KUKA KRL program: MyProgram_195().src

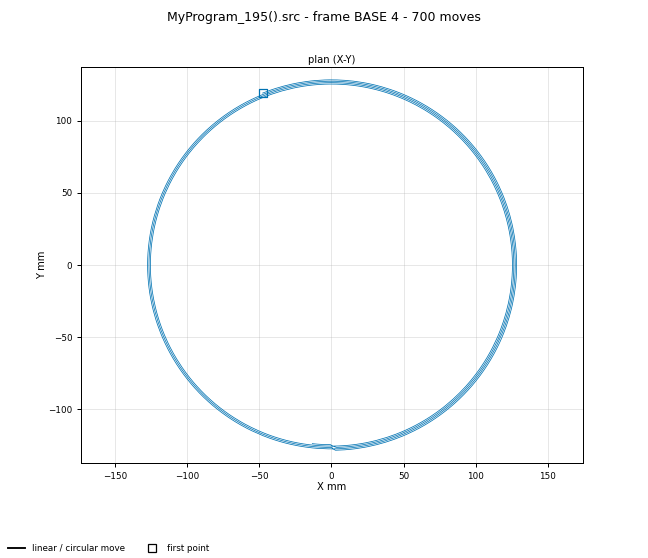
[picture p0: tool path of MyProgram_195().src in frame BASE 4, 700 of 700 moves have a stored position in this frame; points joined in program order, loops and branches not executed]
&ACCESS RVP
&REL 1
&PARAM TEMPLATE = C:\KRC\Roboter\Template\vorgabe
&PARAM EDITMASK = *
DEF MyProgram_195()
; ---- Setting reference (Base) ----
$BASE = BASE_DATA[4]

; --------------------------
; ---- Setting tool (TCP) ----
$TOOL = TOOL_DATA[3]
; --------------------------

$VEL.CP = VEL_APROX_PRINT
Startdeposition()
$VEL.CP = VEL_PRINT
LIN {X -47.6589,Y 119.2143,Z 141,A 107.4986,B 24.9483,C -1.6626,E1 24.9417,E2 698.8654} C_DIS
LIN {X -44.8255,Y 120.308,Z 141,A 106.1446,B 24.9481,C -1.6645,E1 24.9452,E2 700.2177} C_DIS
LIN {X -41.9136,Y 121.3531,Z 141,A 104.7349,B 24.9481,C -1.6649,E1 24.9489,E2 701.6293} C_DIS
LIN {X -38.7242,Y 122.4086,Z 141,A 103.221,B 24.948,C -1.666,E1 24.953,E2 703.1433} C_DIS
LIN {X -35.7429,Y 123.3121,Z 141,A 101.8617,B 24.9478,C -1.669,E1 24.9566,E2 704.4977} C_DIS
LIN {X -32.8744,Y 124.1073,Z 141,A 100.5283,B 24.9478,C -1.6702,E1 24.9602,E2 705.8304} C_DIS
LIN {X -29.3377,Y 124.9928,Z 141,A 98.9078,B 24.9476,C -1.672,E1 24.9646,E2 707.4487} C_DIS
LIN {X -26.9746,Y 125.5218,Z 141,A 97.7935,B 24.9476,C -1.6714,E1 24.9676,E2 708.5658} C_DIS
LIN {X -23.7646,Y 126.1693,Z 141,A 96.3869,B 24.9474,C -1.6752,E1 24.9714,E2 709.965} C_DIS
LIN {X -20.4905,Y 126.7435,Z 141,A 94.8925,B 24.9474,C -1.6758,E1 24.9756,E2 711.4594} C_DIS
LIN {X -17.7576,Y 127.1542,Z 141,A 93.4973,B 24.9478,C -1.6688,E1 24.9795,E2 712.8724} C_DIS
LIN {X -13.7906,Y 127.6448,Z 141,A 91.8165,B 24.9474,C -1.6748,E1 24.9841,E2 714.54} C_DIS
LIN {X -10.7812,Y 127.9341,Z 141,A 90.5046,B 24.9473,C -1.6773,E1 24.9877,E2 715.8467} C_DIS
LIN {X -7.5605,Y 128.1653,Z 141,A 89.0931,B 24.9472,C -1.6793,E1 24.9916,E2 717.254} C_DIS
LIN {X -4.6723,Y 128.3031,Z 141,A 87.7567,B 24.9472,C -1.6775,E1 24.9954,E2 718.5949} C_DIS
LIN {X -1.4217,Y 128.3818,Z 141,A 86.3404,B 24.9472,C -1.6795,E1 24.9993,E2 720.0065} C_DIS
LIN {X 3.8968,Y 128.329,Z 141,A 83.9462,B 24.9472,C -1.6789,E1 25.006,E2 722.4018} C_DIS
LIN {X 6.622,Y 128.2169,Z 141,A 82.776,B 24.947,C -1.6813,E1 25.0093,E2 723.5661} C_DIS
LIN {X 9.4027,Y 128.0429,Z 141,A 81.4527,B 24.9473,C -1.6773,E1 25.013,E2 724.8981} C_DIS
LIN {X 12.4041,Y 127.787,Z 141,A 80.1206,B 24.9473,C -1.6778,E1 25.0167,E2 726.2284} C_DIS
LIN {X 15.3395,Y 127.468,Z 141,A 78.7687,B 24.9473,C -1.6759,E1 25.0204,E2 727.5839} C_DIS
LIN {X 18.503,Y 127.0477,Z 141,A 77.424,B 24.9471,C -1.6794,E1 25.0241,E2 728.919} C_DIS
LIN {X 21.4719,Y 126.5797,Z 141,A 76.0524,B 24.9473,C -1.6774,E1 25.0279,E2 730.2939} C_DIS
LIN {X 25.2565,Y 125.8792,Z 141,A 74.2851,B 24.9475,C -1.6743,E1 25.0328,E2 732.0666} C_DIS
LIN {X 28.5721,Y 125.1677,Z 141,A 72.8026,B 24.9475,C -1.675,E1 25.0368,E2 733.5454} C_DIS
LIN {X 31.6188,Y 124.433,Z 141,A 71.4069,B 24.9475,C -1.6743,E1 25.0406,E2 734.9406} C_DIS
LIN {X 34.9234,Y 123.5467,Z 141,A 69.8932,B 24.9475,C -1.6739,E1 25.0447,E2 736.4528} C_DIS
LIN {X 37.9171,Y 122.661,Z 141,A 68.4959,B 24.9475,C -1.6727,E1 25.0484,E2 737.8507} C_DIS
LIN {X 40.9063,Y 121.6968,Z 141,A 67.0882,B 24.9477,C -1.6712,E1 25.0521,E2 739.2592} C_DIS
LIN {X 43.7241,Y 120.7126,Z 141,A 65.778,B 24.9477,C -1.6711,E1 25.0556,E2 740.567} C_DIS
LIN {X 46.7313,Y 119.5806,Z 141,A 64.3075,B 24.9479,C -1.6678,E1 25.0594,E2 742.042} C_DIS
LIN {X 49.7385,Y 118.3615,Z 141,A 62.882,B 24.9479,C -1.6674,E1 25.0631,E2 743.4652} C_DIS
LIN {X 52.6047,Y 117.1156,Z 141,A 61.4832,B 24.948,C -1.6656,E1 25.0667,E2 744.8649} C_DIS
LIN {X 55.5822,Y 115.7323,Z 141,A 60.0046,B 24.9482,C -1.6631,E1 25.0704,E2 746.3455} C_DIS
LIN {X 58.5789,Y 114.245,Z 141,A 58.5364,B 24.9482,C -1.6624,E1 25.0741,E2 747.8113} C_DIS
LIN {X 61.9613,Y 112.4483,Z 141,A 56.7214,B 24.9487,C -1.6546,E1 25.0786,E2 749.6394} C_DIS
LIN {X 65.8958,Y 110.1886,Z 141,A 54.7394,B 24.9487,C -1.6538,E1 25.0833,E2 751.6175} C_DIS
LIN {X 69.5668,Y 107.9091,Z 141,A 52.8301,B 24.9489,C -1.6517,E1 25.0878,E2 753.5256} C_DIS
LIN {X 72.9887,Y 105.6246,Z 141,A 50.9415,B 24.9492,C -1.6459,E1 25.0922,E2 755.4213} C_DIS
LIN {X 76.5242,Y 103.0914,Z 141,A 49.0479,B 24.9492,C -1.6449,E1 25.0965,E2 757.3107} C_DIS
LIN {X 79.8268,Y 100.5557,Z 141,A 47.1852,B 24.9495,C -1.6412,E1 25.1006,E2 759.1752} C_DIS
LIN {X 83.3011,Y 97.697,Z 141,A 45.1941,B 24.9497,C -1.6381,E1 25.1048,E2 761.1659} C_DIS
LIN {X 86.5812,Y 94.803,Z 141,A 43.2843,B 24.9498,C -1.6363,E1 25.1088,E2 763.0725} C_DIS
LIN {X 89.6025,Y 91.9527,Z 141,A 41.3641,B 24.9503,C -1.6289,E1 25.1127,E2 765.0021} C_DIS
LIN {X 92.6855,Y 88.8435,Z 141,A 39.4441,B 24.9504,C -1.6264,E1 25.1164,E2 766.9199} C_DIS
LIN {X 95.5013,Y 85.8096,Z 141,A 37.6028,B 24.9507,C -1.6224,E1 25.1199,E2 768.7623} C_DIS
LIN {X 98.4786,Y 82.3756,Z 141,A 35.608,B 24.9509,C -1.6194,E1 25.1235,E2 770.7553} C_DIS
LIN {X 101.2232,Y 78.9796,Z 141,A 33.6319,B 24.9512,C -1.6132,E1 25.1269,E2 772.7368} C_DIS
LIN {X 103.8445,Y 75.499,Z 141,A 31.7177,B 24.9514,C -1.6098,E1 25.1301,E2 774.6497} C_DIS
LIN {X 106.4279,Y 71.8114,Z 141,A 29.813,B 24.9514,C -1.6101,E1 25.1331,E2 776.5445} C_DIS
LIN {X 108.4701,Y 68.6878,Z 141,A 28.0658,B 24.9519,C -1.6014,E1 25.1358,E2 778.3034} C_DIS
LIN {X 110.7969,Y 64.8678,Z 141,A 26.1023,B 24.9522,C -1.5976,E1 25.1386,E2 780.2657} C_DIS
LIN {X 112.9064,Y 61.1232,Z 141,A 24.1705,B 24.9525,C -1.5916,E1 25.1412,E2 782.2017} C_DIS
LIN {X 114.6134,Y 57.8552,Z 141,A 22.6765,B 24.9523,C -1.5949,E1 25.1431,E2 783.6799} C_DIS
LIN {X 115.9309,Y 55.1665,Z 141,A 21.3062,B 24.9527,C -1.5893,E1 25.1448,E2 785.0562} C_DIS
LIN {X 117.5259,Y 51.6872,Z 141,A 19.6273,B 24.9529,C -1.5858,E1 25.1467,E2 786.7341} C_DIS
LIN {X 118.5564,Y 49.2718,Z 141,A 18.4452,B 24.9531,C -1.5818,E1 25.148,E2 787.9191} C_DIS
LIN {X 119.7389,Y 46.3239,Z 141,A 17.0649,B 24.9533,C -1.5795,E1 25.1494,E2 789.2971} C_DIS
LIN {X 120.8754,Y 43.2724,Z 141,A 15.6064,B 24.9535,C -1.5749,E1 25.1508,E2 790.7585} C_DIS
LIN {X 121.8283,Y 40.5111,Z 141,A 14.3126,B 24.9537,C -1.5714,E1 25.152,E2 792.0532} C_DIS
LIN {X 122.8365,Y 37.3436,Z 141,A 12.8344,B 24.954,C -1.5671,E1 25.1532,E2 793.5331} C_DIS
LIN {X 123.6826,Y 34.4374,Z 141,A 11.4912,B 24.9542,C -1.5633,E1 25.1542,E2 794.8775} C_DIS
LIN {X 124.4858,Y 31.4106,Z 141,A 10.1044,B 24.9544,C -1.5595,E1 25.1552,E2 796.2653} C_DIS
LIN {X 125.1551,Y 28.6274,Z 141,A 8.8655,B 24.9546,C -1.5575,E1 25.156,E2 797.5018} C_DIS
LIN {X 125.8036,Y 25.6278,Z 141,A 7.4778,B 24.9549,C -1.5522,E1 25.1568,E2 798.8939} C_DIS
LIN {X 126.434,Y 22.3134,Z 141,A 6.0386,B 24.9549,C -1.5509,E1 25.1575,E2 800.3277} C_DIS
LIN {X 126.9286,Y 19.3029,Z 141,A 4.6555,B 24.9553,C -1.5453,E1 25.1581,E2 801.7158} C_DIS
LIN {X 127.3125,Y 16.5798,Z 141,A 3.4224,B 24.9555,C -1.5411,E1 25.1586,E2 802.9517} C_DIS
LIN {X 127.687,Y 13.3981,Z 141,A 1.8638,B 24.9562,C -1.5296,E1 25.1591,E2 804.5281} C_DIS
LIN {X 128.0429,Y 9.4019,Z 141,A 0.2073,B 24.9561,C -1.5308,E1 25.1594,E2 806.1719} C_DIS
LIN {X 128.262,Y 5.7236,Z 141,A -1.3842,B 24.9562,C -1.5282,E1 25.1597,E2 807.7601} C_DIS
LIN {X 128.3645,Y 2.4644,Z 141,A -2.6743,B 24.956,C -1.5322,E1 25.1597,E2 809.0331} C_DIS
LIN {X 128.3668,Y -2.3216,Z 141,A -4.9685,B 24.9569,C -1.5168,E1 25.1597,E2 811.35} C_DIS
LIN {X 128.262,Y -5.7236,Z 141,A -6.4603,B 24.9571,C -1.5132,E1 25.1596,E2 812.8414} C_DIS
LIN {X 128.1,Y -8.6199,Z 141,A -7.7483,B 24.9573,C -1.5092,E1 25.1594,E2 814.131} C_DIS
LIN {X 127.828,Y -11.978,Z 141,A -9.3108,B 24.9578,C -1.5012,E1 25.159,E2 815.7033} C_DIS
LIN {X 127.4547,Y -15.4503,Z 141,A -10.7633,B 24.9578,C -1.5016,E1 25.1585,E2 817.1461} C_DIS
LIN {X 127.0477,Y -18.503,Z 141,A -12.1966,B 24.9582,C -1.494,E1 25.158,E2 818.589} C_DIS
LIN {X 126.5797,Y -21.4719,Z 141,A -13.5133,B 24.9584,C -1.4909,E1 25.1574,E2 819.9053} C_DIS
LIN {X 126.1015,Y -24.1193,Z 141,A -14.7002,B 24.9585,C -1.4877,E1 25.1568,E2 821.0928} C_DIS
LIN {X 125.448,Y -27.3165,Z 141,A -16.1278,B 24.9587,C -1.4844,E1 25.156,E2 822.5196} C_DIS
LIN {X 124.7294,Y -30.4307,Z 141,A -17.5353,B 24.9589,C -1.4808,E1 25.1551,E2 823.9276} C_DIS
LIN {X 123.9197,Y -33.5779,Z 141,A -18.989,B 24.9592,C -1.4759,E1 25.154,E2 825.3844} C_DIS
LIN {X 123.0744,Y -36.5547,Z 141,A -20.3562,B 24.9594,C -1.4722,E1 25.153,E2 826.7527} C_DIS
LIN {X 122.2177,Y -39.3218,Z 141,A -21.6718,B 24.9597,C -1.4668,E1 25.1518,E2 828.0734} C_DIS
LIN {X 121.2238,Y -42.2863,Z 141,A -23.1033,B 24.96,C -1.4604,E1 25.1505,E2 829.5118} C_DIS
LIN {X 119.5855,Y -46.7186,Z 141,A -25.1701,B 24.9603,C -1.456,E1 25.1485,E2 831.5775} C_DIS
LIN {X 118.3511,Y -49.7632,Z 141,A -26.6151,B 24.9605,C -1.4525,E1 25.147,E2 833.0228} C_DIS
LIN {X 117.0468,Y -52.7584,Z 141,A -28.0533,B 24.9607,C -1.4491,E1 25.1453,E2 834.4614} C_DIS
LIN {X 115.6855,Y -55.6801,Z 141,A -29.4664,B 24.9608,C -1.446,E1 25.1437,E2 835.8741} C_DIS
LIN {X 114.245,Y -58.5789,Z 141,A -30.9204,B 24.9611,C -1.4411,E1 25.1418,E2 837.3319} C_DIS
LIN {X 112.5421,Y -61.7911,Z 141,A -32.6609,B 24.9617,C -1.4299,E1 25.1395,E2 839.0895} C_DIS
LIN {X 110.4276,Y -65.4948,Z 141,A -34.5555,B 24.962,C -1.4248,E1 25.1368,E2 840.9866} C_DIS
LIN {X 108.0286,Y -69.3801,Z 141,A -36.5281,B 24.9621,C -1.4223,E1 25.1339,E2 842.9551} C_DIS
LIN {X 105.6246,Y -72.9887,Z 141,A -38.5037,B 24.9625,C -1.4146,E1 25.1308,E2 844.939} C_DIS
LIN {X 103.0914,Y -76.5242,Z 141,A -40.4163,B 24.9627,C -1.4107,E1 25.1276,E2 846.8516} C_DIS
LIN {X 100.3351,Y -80.104,Z 141,A -42.3438,B 24.9627,C -1.4098,E1 25.1243,E2 848.772} C_DIS
LIN {X 97.697,Y -83.3011,Z 141,A -44.2446,B 24.9632,C -1.4022,E1 25.1209,E2 850.6821} C_DIS
LIN {X 94.803,Y -86.5812,Z 141,A -46.1541,B 24.9633,C -1.3993,E1 25.1174,E2 852.5898} C_DIS
LIN {X 91.9527,Y -89.6025,Z 141,A -48.0782,B 24.9638,C -1.3909,E1 25.1136,E2 854.5255} C_DIS
LIN {X 88.8435,Y -92.6855,Z 141,A -49.9915,B 24.9638,C -1.3883,E1 25.1098,E2 856.4371} C_DIS
LIN {X 85.5442,Y -95.739,Z 141,A -51.9159,B 24.9639,C -1.3877,E1 25.1058,E2 858.3549} C_DIS
LIN {X 82.4171,Y -98.4438,Z 141,A -53.799,B 24.9643,C -1.3815,E1 25.1018,E2 860.2454} C_DIS
LIN {X 78.9796,Y -101.2232,Z 141,A -55.8093,B 24.9646,C -1.3751,E1 25.0974,E2 862.2633} C_DIS
LIN {X 75.5335,Y -103.8195,Z 141,A -57.7116,B 24.9647,C -1.3722,E1 25.0931,E2 864.1657} C_DIS
LIN {X 71.8114,Y -106.4279,Z 141,A -59.642,B 24.9647,C -1.3731,E1 25.0887,E2 866.0873} C_DIS
LIN {X 68.6878,Y -108.4701,Z 141,A -61.3769,B 24.965,C -1.3662,E1 25.0846,E2 867.8328} C_DIS
LIN {X 64.8678,Y -110.7969,Z 141,A -63.3553,B 24.9652,C -1.3634,E1 25.0799,E2 869.8119} C_DIS
LIN {X 61.0702,Y -112.935,Z 141,A -65.3382,B 24.9655,C -1.3579,E1 25.075,E2 871.8018} C_DIS
LIN {X 57.524,Y -114.782,Z 141,A -66.9688,B 24.9652,C -1.3628,E1 25.071,E2 873.4165} C_DIS
LIN {X 54.8837,Y -116.0659,Z 141,A -68.2914,B 24.9654,C -1.36,E1 25.0677,E2 874.7422} C_DIS
LIN {X 52.194,Y -117.2993,Z 141,A -69.6034,B 24.9654,C -1.3584,E1 25.0643,E2 876.0547} C_DIS
LIN {X 49.1377,Y -118.6124,Z 141,A -71.057,B 24.9654,C -1.3578,E1 25.0606,E2 877.5064} C_DIS
LIN {X 46.2845,Y -119.7543,Z 141,A -72.4524,B 24.9656,C -1.3546,E1 25.057,E2 878.9061} C_DIS
LIN {X 43.3744,Y -120.8386,Z 141,A -73.8237,B 24.9656,C -1.3535,E1 25.0534,E2 880.2772} C_DIS
LIN {X 40.218,Y -121.926,Z 141,A -75.296,B 24.9657,C -1.3525,E1 25.0495,E2 881.7491} C_DIS
LIN {X 37.3931,Y -122.8214,Z 141,A -76.6369,B 24.9659,C -1.35,E1 25.0459,E2 883.0936} C_DIS
LIN {X 33.9807,Y -123.8104,Z 141,A -78.1804,B 24.9659,C -1.3503,E1 25.0417,E2 884.6336} C_DIS
LIN {X 31.2387,Y -124.5295,Z 141,A -79.4595,B 24.9659,C -1.3483,E1 25.0383,E2 885.9155} C_DIS
LIN {X 28.2554,Y -125.2401,Z 141,A -80.8337,B 24.966,C -1.3467,E1 25.0345,E2 887.2916} C_DIS
LIN {X 25.3982,Y -125.8503,Z 141,A -82.0646,B 24.966,C -1.3492,E1 25.0312,E2 888.5151} C_DIS
LIN {X 22.6034,Y -126.3821,Z 141,A -83.3984,B 24.9661,C -1.3449,E1 25.0275,E2 889.8575} C_DIS
LIN {X 19.3029,Y -126.9286,Z 141,A -84.8397,B 24.9661,C -1.3464,E1 25.0235,E2 891.2939} C_DIS
LIN {X 16.5401,Y -127.3177,Z 141,A -86.1724,B 24.9663,C -1.3411,E1 25.0198,E2 892.6379} C_DIS
LIN {X 13.3981,Y -127.687,Z 141,A -87.5525,B 24.9663,C -1.3419,E1 25.016,E2 894.0153} C_DIS
LIN {X 9.3263,Y -128.0484,Z 141,A -89.3875,B 24.9663,C -1.3404,E1 25.0109,E2 895.8527} C_DIS
LIN {X 5.7236,Y -128.262,Z 141,A -90.9441,B 24.9663,C -1.3425,E1 25.0066,E2 897.4039} C_DIS
LIN {X 2.8497,Y -128.3581,Z 141,A -92.2242,B 24.9663,C -1.3422,E1 25.003,E2 898.6844} C_DIS
LIN {X 2.8497,Y -128.3581,Z 141,A -92.2242,B 24.9663,C -1.3422,E1 25.003,E2 898.6844} C_DIS
Enddeposition()
LIN {X 0.8999,Y -127.3905,Z 141,A -92.6866,B 24.9643,C -1.3799,E1 25.0019,E2 899.0576} C_DIS
Startdeposition()
$VEL.CP = VEL_PRINT
LIN {X 5.0187,Y -127.3169,Z 141,A -90.0531,B 24.9623,C -1.4196,E1 25.0096,E2 896.3305} C_DIS
LIN {X 9.7195,Y -127.0453,Z 141,A -88.5298,B 24.9638,C -1.3904,E1 25.0136,E2 894.8772} C_DIS
LIN {X 13.7182,Y -126.6751,Z 141,A -86.6564,B 24.9636,C -1.3948,E1 25.0188,E2 892.9945} C_DIS
LIN {X 17.7849,Y -126.1685,Z 141,A -84.8963,B 24.9637,C -1.3918,E1 25.0237,E2 891.2428} C_DIS
LIN {X 21.0971,Y -125.6569,Z 141,A -83.3739,B 24.9637,C -1.3937,E1 25.0279,E2 889.7174} C_DIS
LIN {X 25.0147,Y -124.9366,Z 141,A -81.5858,B 24.9635,C -1.3951,E1 25.0328,E2 887.9282} C_DIS
LIN {X 28.3959,Y -124.2111,Z 141,A -80.043,B 24.9635,C -1.3959,E1 25.037,E2 886.3855} C_DIS
LIN {X 31.7595,Y -123.3946,Z 141,A -78.3701,B 24.9631,C -1.4035,E1 25.0416,E2 884.6972} C_DIS
LIN {X 36.6091,Y -122.0449,Z 141,A -76.1613,B 24.9631,C -1.4032,E1 25.0475,E2 882.4928} C_DIS
LIN {X 43.7793,Y -119.6595,Z 141,A -72.714,B 24.9628,C -1.4101,E1 25.0566,E2 879.036} C_DIS
LIN {X 49.8999,Y -117.2399,Z 141,A -69.8104,B 24.9627,C -1.4115,E1 25.0641,E2 876.1358} C_DIS
LIN {X 53.3784,Y -115.6954,Z 141,A -68.1964,B 24.9628,C -1.4092,E1 25.0682,E2 874.5312} C_DIS
LIN {X 57.1272,Y -113.8934,Z 141,A -66.2114,B 24.9623,C -1.4182,E1 25.0732,E2 872.5302} C_DIS
LIN {X 60.7457,Y -112.0053,Z 141,A -64.4039,B 24.9623,C -1.4199,E1 25.0777,E2 870.7237} C_DIS
LIN {X 64.419,Y -109.9334,Z 141,A -62.5287,B 24.9621,C -1.4223,E1 25.0822,E2 868.8486} C_DIS
LIN {X 67.7995,Y -107.8815,Z 141,A -60.3446,B 24.9608,C -1.447,E1 25.0875,E2 866.613} C_DIS
LIN {X 71.2712,Y -105.62,Z 141,A -58.8855,B 24.9617,C -1.4296,E1 25.0908,E2 865.2} C_DIS
LIN {X 74.9106,Y -103.0706,Z 141,A -56.9736,B 24.9617,C -1.4293,E1 25.0951,E2 863.2955} C_DIS
LIN {X 78.716,Y -100.1944,Z 141,A -54.7473,B 24.9613,C -1.4382,E1 25.1001,E2 861.0562} C_DIS
LIN {X 82.1169,Y -97.427,Z 141,A -52.81,B 24.9611,C -1.4409,E1 25.1042,E2 859.12} C_DIS
LIN {X 85.144,Y -94.7927,Z 141,A -51.0136,B 24.9609,C -1.4447,E1 25.108,E2 857.3217} C_DIS
LIN {X 88.5702,Y -91.5995,Z 141,A -48.8304,B 24.9604,C -1.4539,E1 25.1124,E2 855.1258} C_DIS
LIN {X 91.8325,Y -88.3294,Z 141,A -46.8129,B 24.9603,C -1.456,E1 25.1164,E2 853.112} C_DIS
LIN {X 94.6423,Y -85.3119,Z 141,A -45.2051,B 24.9607,C -1.4478,E1 25.1194,E2 851.5306} C_DIS
LIN {X 97.0825,Y -82.5234,Z 141,A -43.1322,B 24.9593,C -1.4737,E1 25.1232,E2 849.4061} C_DIS
LIN {X 99.1334,Y -80.0482,Z 141,A -41.8163,B 24.9595,C -1.4708,E1 25.1255,E2 848.1032} C_DIS
LIN {X 102.0489,Y -76.2968,Z 141,A -39.7646,B 24.9594,C -1.4722,E1 25.129,E2 846.058} C_DIS
LIN {X 103.7413,Y -73.9791,Z 141,A -37.7936,B 24.9572,C -1.5121,E1 25.1323,E2 844.0024} C_DIS
LIN {X 106.9396,Y -69.2754,Z 141,A -36.0227,B 24.9591,C -1.4774,E1 25.1349,E2 842.3222} C_DIS
LIN {X 109.1238,Y -65.7811,Z 141,A -34.1648,B 24.9588,C -1.4831,E1 25.1376,E2 840.4603} C_DIS
LIN {X 111.2174,Y -62.1765,Z 141,A -32.2654,B 24.9584,C -1.49,E1 25.1402,E2 838.5546} C_DIS
LIN {X 113.327,Y -58.2398,Z 141,A -30.3103,B 24.9582,C -1.4932,E1 25.1428,E2 836.6021} C_DIS
LIN {X 114.7515,Y -55.3804,Z 141,A -28.6393,B 24.9573,C -1.5101,E1 25.1448,E2 834.9002} C_DIS
LIN {X 118.1649,Y -47.6626,Z 141,A -25.099,B 24.9573,C -1.5083,E1 25.1487,E2 831.3836} C_DIS
LIN {X 119.4462,Y -44.3549,Z 141,A -23.4481,B 24.9569,C -1.5163,E1 25.1503,E2 829.7229} C_DIS
LIN {X 120.853,Y -40.364,Z 141,A -21.6913,B 24.957,C -1.5146,E1 25.1519,E2 827.9801} C_DIS
LIN {X 122.1027,Y -36.4146,Z 141,A -19.7328,B 24.9564,C -1.5257,E1 25.1535,E2 826.0067} C_DIS
LIN {X 123.0116,Y -33.2114,Z 141,A -18.2861,B 24.9563,C -1.5278,E1 25.1546,E2 824.5632} C_DIS
LIN {X 123.9321,Y -29.5908,Z 141,A -16.6689,B 24.9561,C -1.53,E1 25.1557,E2 822.9504} C_DIS
LIN {X 124.9603,Y -24.8983,Z 141,A -14.406,B 24.9554,C -1.5425,E1 25.157,E2 820.6711} C_DIS
LIN {X 125.6731,Y -20.9999,Z 141,A -12.734,B 24.9554,C -1.5425,E1 25.1578,E2 819.0089} C_DIS
LIN {X 126.2869,Y -16.9267,Z 141,A -10.888,B 24.9551,C -1.5482,E1 25.1585,E2 817.1603} C_DIS
LIN {X 126.7017,Y -13.4706,Z 141,A -9.3374,B 24.9548,C -1.5526,E1 25.159,E2 815.6085} C_DIS
LIN {X 127.07,Y -9.38,Z 141,A -7.5103,B 24.9545,C -1.5577,E1 25.1594,E2 813.7803} C_DIS
LIN {X 127.304,Y -5.3489,Z 141,A -5.6211,B 24.954,C -1.5676,E1 25.1597,E2 811.879} C_DIS
LIN {X 127.4162,Y -0.6084,Z 141,A -3.557,B 24.9538,C -1.5709,E1 25.1597,E2 809.8193} C_DIS
LIN {X 127.3666,Y 3.5418,Z 141,A -1.7145,B 24.9535,C -1.5758,E1 25.1597,E2 807.9762} C_DIS
LIN {X 127.1779,Y 7.7828,Z 141,A 0.1626,B 24.9532,C -1.5804,E1 25.1594,E2 806.0995} C_DIS
LIN {X 126.8599,Y 11.8919,Z 141,A 2.0078,B 24.9529,C -1.586,E1 25.159,E2 804.252} C_DIS
LIN {X 126.4848,Y 15.3762,Z 141,A 3.6561,B 24.9523,C -1.595,E1 25.1584,E2 802.5923} C_DIS
LIN {X 125.9688,Y 19.1503,Z 141,A 5.3086,B 24.9522,C -1.5973,E1 25.1578,E2 800.9441} C_DIS
LIN {X 125.3635,Y 22.7779,Z 141,A 6.9826,B 24.9518,C -1.6037,E1 25.157,E2 799.2649} C_DIS
LIN {X 124.558,Y 26.8331,Z 141,A 8.757,B 24.9518,C -1.6051,E1 25.156,E2 797.4974} C_DIS
LIN {X 123.6768,Y 30.6475,Z 141,A 10.5659,B 24.9512,C -1.6132,E1 25.1548,E2 795.68} C_DIS
LIN {X 122.7672,Y 34.1021,Z 141,A 12.0916,B 24.9512,C -1.6139,E1 25.1537,E2 794.1612} C_DIS
LIN {X 120.3644,Y 41.7982,Z 141,A 15.669,B 24.9507,C -1.6225,E1 25.1507,E2 790.584} C_DIS
LIN {X 118.2298,Y 47.5016,Z 141,A 18.3975,B 24.9502,C -1.6301,E1 25.1479,E2 787.8526} C_DIS
LIN {X 117.0733,Y 50.2852,Z 141,A 19.7851,B 24.9499,C -1.6358,E1 25.1464,E2 786.4593} C_DIS
LIN {X 115.6821,Y 53.407,Z 141,A 21.2613,B 24.9498,C -1.6371,E1 25.1447,E2 784.988} C_DIS
LIN {X 113.6179,Y 57.6684,Z 141,A 23.3544,B 24.9495,C -1.6413,E1 25.1421,E2 782.8963} C_DIS
LIN {X 111.966,Y 60.8178,Z 141,A 25.092,B 24.9488,C -1.653,E1 25.1398,E2 781.1402} C_DIS
LIN {X 110.3693,Y 63.6693,Z 141,A 26.6703,B 24.9482,C -1.6628,E1 25.1376,E2 779.547} C_DIS
LIN {X 107.8529,Y 67.8448,Z 141,A 28.7103,B 24.9483,C -1.6607,E1 25.1346,E2 777.5223} C_DIS
LIN {X 105.5211,Y 71.4173,Z 141,A 31.4001,B 24.9454,C -1.7064,E1 25.1303,E2 774.7379} C_DIS
LIN {X 102.032,Y 76.3196,Z 141,A 33.1048,B 24.9483,C -1.6606,E1 25.1277,E2 773.1496} C_DIS
LIN {X 99.6963,Y 79.3459,Z 141,A 35.0176,B 24.9474,C -1.6749,E1 25.1243,E2 771.212} C_DIS
LIN {X 96.8479,Y 82.7994,Z 141,A 37.0608,B 24.947,C -1.6813,E1 25.1206,E2 769.163} C_DIS
LIN {X 94.0234,Y 85.9932,Z 141,A 38.9764,B 24.9468,C -1.6856,E1 25.117,E2 767.2458} C_DIS
LIN {X 90.9534,Y 89.2335,Z 141,A 40.9351,B 24.9466,C -1.6876,E1 25.1133,E2 765.2909} C_DIS
LIN {X 87.7985,Y 92.3399,Z 141,A 42.9285,B 24.9464,C -1.6919,E1 25.1093,E2 763.2955} C_DIS
LIN {X 84.6166,Y 95.2641,Z 141,A 44.8865,B 24.9461,C -1.6967,E1 25.1052,E2 761.334} C_DIS
LIN {X 82.3184,Y 97.2568,Z 141,A 47.3402,B 24.9422,C -1.7559,E1 25.0997,E2 758.7499} C_DIS
LIN {X 76.2571,Y 102.0785,Z 141,A 49.3622,B 24.9467,C -1.6865,E1 25.0956,E2 756.8992} C_DIS
LIN {X 73.2603,Y 104.2502,Z 141,A 51.3498,B 24.9455,C -1.706,E1 25.091,E2 754.8727} C_DIS
LIN {X 69.6579,Y 106.6912,Z 141,A 53.3231,B 24.9452,C -1.7101,E1 25.0863,E2 752.8963} C_DIS
LIN {X 66.2943,Y 108.8133,Z 141,A 55.1701,B 24.9448,C -1.7158,E1 25.0819,E2 751.0414} C_DIS
LIN {X 62.1147,Y 111.2521,Z 141,A 57.2696,B 24.9448,C -1.7151,E1 25.0769,E2 748.95} C_DIS
LIN {X 58.4758,Y 113.2069,Z 141,A 58.9718,B 24.9452,C -1.7097,E1 25.0727,E2 747.2652} C_DIS
LIN {X 55.396,Y 114.7441,Z 141,A 60.6108,B 24.9448,C -1.7163,E1 25.0686,E2 745.6149} C_DIS
LIN {X 52.311,Y 116.1822,Z 141,A 62.0976,B 24.9448,C -1.716,E1 25.0648,E2 744.1328} C_DIS
LIN {X 49.3995,Y 117.4498,Z 141,A 64.2393,B 24.9424,C -1.7538,E1 25.0591,E2 741.9067} C_DIS
LIN {X 44.4245,Y 119.4203,Z 141,A 65.9616,B 24.9445,C -1.7214,E1 25.0548,E2 740.2647} C_DIS
LIN {X 39.2905,Y 121.2074,Z 141,A 68.4163,B 24.9443,C -1.724,E1 25.0483,E2 737.8085} C_DIS
LIN {X 35.769,Y 122.2918,Z 141,A 70.003,B 24.9444,C -1.7218,E1 25.0441,E2 736.23} C_DIS
LIN {X 32.056,Y 123.3193,Z 141,A 71.8461,B 24.944,C -1.7284,E1 25.0391,E2 734.3741} C_DIS
LIN {X 28.4356,Y 124.202,Z 141,A 73.339,B 24.9445,C -1.7203,E1 25.0351,E2 732.9025} C_DIS
LIN {X 24.8772,Y 124.9646,Z 141,A 75.1472,B 24.9439,C -1.7296,E1 25.0301,E2 731.0746} C_DIS
LIN {X 21.0816,Y 125.6595,Z 141,A 76.7751,B 24.9442,C -1.7249,E1 25.0256,E2 729.4594} C_DIS
LIN {X 17.3933,Y 126.2245,Z 141,A 78.5767,B 24.9438,C -1.7315,E1 25.0206,E2 727.644} C_DIS
LIN {X 13.5608,Y 126.692,Z 141,A 80.2111,B 24.9441,C -1.7268,E1 25.0161,E2 726.0219} C_DIS
LIN {X 9.3897,Y 127.0693,Z 141,A 82.0663,B 24.9441,C -1.7255,E1 25.0109,E2 724.1706} C_DIS
LIN {X 5.6118,Y 127.2938,Z 141,A 83.8503,B 24.9439,C -1.7295,E1 25.0059,E2 722.3778} C_DIS
LIN {X 1.9512,Y 127.401,Z 141,A 85.5028,B 24.9439,C -1.7295,E1 25.0013,E2 720.7254} C_DIS
LIN {X -2.0548,Y 127.3993,Z 141,A 87.2207,B 24.9442,C -1.7251,E1 24.9966,E2 719.0181} C_DIS
LIN {X -5.8827,Y 127.2809,Z 141,A 89.0271,B 24.944,C -1.7286,E1 24.9915,E2 717.2029} C_DIS
LIN {X -9.8951,Y 127.0324,Z 141,A 90.8694,B 24.944,C -1.7296,E1 24.9864,E2 715.3578} C_DIS
LIN {X -13.7094,Y 126.676,Z 141,A 92.4979,B 24.9443,C -1.7241,E1 24.9819,E2 713.7413} C_DIS
LIN {X -17.7756,Y 126.1699,Z 141,A 94.3454,B 24.9443,C -1.7232,E1 24.9768,E2 711.8946} C_DIS
LIN {X -21.2439,Y 125.6324,Z 141,A 96.0119,B 24.9441,C -1.7263,E1 24.9721,E2 710.2191} C_DIS
LIN {X -25.6157,Y 124.8143,Z 141,A 98.1557,B 24.9438,C -1.7316,E1 24.9662,E2 708.0603} C_DIS
LIN {X -30.2633,Y 123.77,Z 141,A 100.1654,B 24.9444,C -1.7232,E1 24.9608,E2 706.0679} C_DIS
LIN {X -34.1946,Y 122.7414,Z 141,A 101.8446,B 24.9449,C -1.7142,E1 24.9563,E2 704.4076} C_DIS
LIN {X -40.9405,Y 120.661,Z 141,A 105.0429,B 24.9451,C -1.7115,E1 24.9478,E2 701.21} C_DIS
LIN {X -45.8326,Y 118.8872,Z 141,A 107.426,B 24.9451,C -1.7104,E1 24.9416,E2 698.8244} C_DIS
LIN {X -49.0691,Y 117.5878,Z 141,A 108.8652,B 24.9457,C -1.7021,E1 24.9379,E2 697.4019} C_DIS
LIN {X -51.8592,Y 116.3843,Z 141,A 110.4026,B 24.9453,C -1.7082,E1 24.9339,E2 695.8464} C_DIS
LIN {X -55.4111,Y 114.7369,Z 141,A 112.2581,B 24.9453,C -1.7099,E1 24.9292,E2 693.9822} C_DIS
LIN {X -58.8494,Y 113.0114,Z 141,A 113.8944,B 24.9457,C -1.7025,E1 24.9252,E2 692.3589} C_DIS
LIN {X -62.7237,Y 110.9098,Z 141,A 116.1068,B 24.9452,C -1.7099,E1 24.9197,E2 690.1225} C_DIS
LIN {X -66.9445,Y 108.4145,Z 141,A 118.1975,B 24.9458,C -1.7004,E1 24.9148,E2 688.048} C_DIS
LIN {X -70.7251,Y 105.9863,Z 141,A 120.1943,B 24.9461,C -1.6953,E1 24.9101,E2 686.0568} C_DIS
LIN {X -74.4535,Y 103.4019,Z 141,A 122.2733,B 24.9463,C -1.6929,E1 24.9054,E2 683.9763} C_DIS
LIN {X -78.0433,Y 100.7192,Z 141,A 124.2429,B 24.9467,C -1.6865,E1 24.901,E2 682.015} C_DIS
LIN {X -82.094,Y 97.4462,Z 141,A 126.8108,B 24.9464,C -1.6918,E1 24.8954,E2 679.4246} C_DIS
LIN {X -86.2732,Y 93.766,Z 141,A 129.1169,B 24.9473,C -1.6767,E1 24.8907,E2 677.1452} C_DIS
LIN {X -89.5721,Y 90.6205,Z 141,A 131.1797,B 24.9476,C -1.6723,E1 24.8866,E2 675.0843} C_DIS
LIN {X -92.5001,Y 87.6295,Z 141,A 133.0568,B 24.9479,C -1.6673,E1 24.8829,E2 673.2109} C_DIS
LIN {X -95.2867,Y 84.591,Z 141,A 134.9703,B 24.948,C -1.6653,E1 24.8794,E2 671.2936} C_DIS
LIN {X -98.2414,Y 81.1405,Z 141,A 136.9783,B 24.9485,C -1.6583,E1 24.8758,E2 669.2931} C_DIS
LIN {X -100.962,Y 77.7301,Z 141,A 139.0197,B 24.9485,C -1.6567,E1 24.8722,E2 667.246} C_DIS
LIN {X -103.6546,Y 74.1003,Z 141,A 140.9864,B 24.9491,C -1.648,E1 24.869,E2 665.2903} C_DIS
LIN {X -106.1366,Y 70.5,Z 141,A 143.011,B 24.9493,C -1.6451,E1 24.8659,E2 663.2626} C_DIS
LIN {X -108.4427,Y 66.8986,Z 141,A 144.8042,B 24.95,C -1.6336,E1 24.8632,E2 661.4878} C_DIS
LIN {X -111.4259,Y 61.8013,Z 141,A 147.5817,B 24.9501,C -1.6314,E1 24.8593,E2 658.7012} C_DIS
LIN {X -113.4093,Y 58.0782,Z 141,A 149.4329,B 24.9506,C -1.6236,E1 24.8569,E2 656.8586} C_DIS
LIN {X -114.8825,Y 55.1063,Z 141,A 150.9228,B 24.9509,C -1.619,E1 24.8551,E2 655.3716} C_DIS
LIN {X -117.221,Y 49.9435,Z 141,A 153.6361,B 24.9509,C -1.6186,E1 24.8521,E2 652.6442} C_DIS
LIN {X -118.9475,Y 45.6774,Z 141,A 155.6993,B 24.9513,C -1.6119,E1 24.8499,E2 650.5855} C_DIS
LIN {X -120.3282,Y 41.9028,Z 141,A 157.3907,B 24.952,C -1.6008,E1 24.8484,E2 648.9109} C_DIS
LIN {X -122.72,Y 34.2709,Z 141,A 160.9993,B 24.9526,C -1.5898,E1 24.8454,E2 645.3078} C_DIS
LIN {X -123.9277,Y 29.6091,Z 141,A 163.2602,B 24.9528,C -1.5872,E1 24.8439,E2 643.0399} C_DIS
LIN {X -124.7694,Y 25.8361,Z 141,A 165.0561,B 24.953,C -1.5841,E1 24.8428,E2 641.2407} C_DIS
LIN {X -125.559,Y 21.6838,Z 141,A 166.9904,B 24.9533,C -1.5795,E1 24.8419,E2 639.3061} C_DIS
LIN {X -126.2524,Y 17.1897,Z 141,A 169.136,B 24.9533,C -1.5774,E1 24.841,E2 637.1526} C_DIS
LIN {X -126.8159,Y 12.3501,Z 141,A 171.1416,B 24.9543,C -1.5617,E1 24.8404,E2 635.1725} C_DIS
LIN {X -127.1382,Y 8.4266,Z 141,A 172.9805,B 24.9545,C -1.559,E1 24.8401,E2 633.3289} C_DIS
LIN {X -127.3292,Y 4.703,Z 141,A 174.7074,B 24.9546,C -1.5558,E1 24.8398,E2 631.5993} C_DIS
LIN {X -127.418,Y 0.298,Z 141,A 176.7523,B 24.9549,C -1.5522,E1 24.8398,E2 629.5506} C_DIS
LIN {X -127.3609,Y -3.7471,Z 141,A 178.4593,B 24.9555,C -1.5411,E1 24.8398,E2 627.8598} C_DIS
LIN {X -127.1848,Y -7.6702,Z 141,A -179.7545,B 24.9558,C -1.5362,E1 24.8402,E2 626.0744} C_DIS
LIN {X -126.8768,Y -11.716,Z 141,A -177.9197,B 24.9561,C -1.5308,E1 24.8406,E2 624.2417} C_DIS
LIN {X -126.4648,Y -15.5439,Z 141,A -176.1542,B 24.9563,C -1.5267,E1 24.8412,E2 622.4752} C_DIS
LIN {X -125.9319,Y -19.3887,Z 141,A -174.5801,B 24.9571,C -1.5132,E1 24.8418,E2 620.9238} C_DIS
LIN {X -125.3697,Y -22.7433,Z 141,A -172.9329,B 24.9571,C -1.5137,E1 24.8426,E2 619.2656} C_DIS
LIN {X -124.2875,Y -28.0612,Z 141,A -170.4309,B 24.9573,C -1.5088,E1 24.844,E2 616.7607} C_DIS
LIN {X -123.484,Y -31.4073,Z 141,A -168.886,B 24.9576,C -1.5039,E1 24.8451,E2 615.2185} C_DIS
LIN {X -121.6554,Y -37.8819,Z 141,A -165.7394,B 24.9578,C -1.5001,E1 24.8475,E2 612.0628} C_DIS
LIN {X -120.4598,Y -41.523,Z 141,A -164.2093,B 24.9586,C -1.4859,E1 24.8489,E2 610.5577} C_DIS
LIN {X -119.3853,Y -44.5182,Z 141,A -162.6888,B 24.9586,C -1.4857,E1 24.8503,E2 609.029} C_DIS
LIN {X -118.2732,Y -47.394,Z 141,A -161.304,B 24.9589,C -1.4815,E1 24.8517,E2 607.6465} C_DIS
LIN {X -117.0082,Y -50.4358,Z 141,A -159.7841,B 24.959,C -1.479,E1 24.8534,E2 606.1243} C_DIS
LIN {X -115.5315,Y -53.7327,Z 141,A -157.5953,B 24.9578,C -1.5007,E1 24.8561,E2 603.8718} C_DIS
LIN {X -113.5646,Y -57.7731,Z 141,A -156.14,B 24.9596,C -1.4684,E1 24.8578,E2 602.4856} C_DIS
LIN {X -111.8885,Y -60.9598,Z 141,A -154.4185,B 24.9596,C -1.4686,E1 24.8601,E2 600.7544} C_DIS
LIN {X -109.6733,Y -64.8617,Z 141,A -152.346,B 24.9598,C -1.4657,E1 24.863,E2 598.6782} C_DIS
LIN {X -107.465,Y -68.4579,Z 141,A -150.4482,B 24.96,C -1.4606,E1 24.8658,E2 596.7827} C_DIS
LIN {X -104.9915,Y -72.1937,Z 141,A -148.4483,B 24.9604,C -1.4547,E1 24.8689,E2 594.787} C_DIS
LIN {X -102.4469,Y -75.7623,Z 141,A -146.4367,B 24.9605,C -1.4516,E1 24.8722,E2 592.773} C_DIS
LIN {X -99.8054,Y -79.2089,Z 141,A -144.5042,B 24.9608,C -1.4459,E1 24.8755,E2 590.8449} C_DIS
LIN {X -97.0404,Y -82.573,Z 141,A -142.5342,B 24.9611,C -1.4418,E1 24.8791,E2 588.8756} C_DIS
LIN {X -94.6485,Y -85.3049,Z 141,A -140.85,B 24.9611,C -1.4404,E1 24.8822,E2 587.1872} C_DIS
LIN {X -91.6526,Y -88.5153,Z 141,A -138.9105,B 24.9615,C -1.4344,E1 24.8859,E2 585.2537} C_DIS
LIN {X -88.4976,Y -91.6697,Z 141,A -136.9516,B 24.9618,C -1.4278,E1 24.8898,E2 583.3021} C_DIS
LIN {X -85.3862,Y -94.575,Z 141,A -134.9806,B 24.9618,C -1.4266,E1 24.8939,E2 581.326} C_DIS
LIN {X -82.2202,Y -97.3403,Z 141,A -133.0502,B 24.962,C -1.4248,E1 24.898,E2 579.3924} C_DIS
LIN {X -78.8653,Y -100.0772,Z 141,A -131.1475,B 24.9623,C -1.419,E1 24.9021,E2 577.4963} C_DIS
LIN {X -75.7193,Y -102.4785,Z 141,A -129.295,B 24.9623,C -1.4193,E1 24.9062,E2 575.6366} C_DIS
LIN {X -72.0276,Y -105.1054,Z 141,A -127.2955,B 24.9625,C -1.414,E1 24.9108,E2 573.6427} C_DIS
LIN {X -69.3367,Y -106.8998,Z 141,A -125.5913,B 24.962,C -1.4238,E1 24.9149,E2 571.9099} C_DIS
LIN {X -66.5217,Y -108.6739,Z 141,A -124.3577,B 24.9628,C -1.4088,E1 24.9177,E2 570.7081} C_DIS
LIN {X -62.879,Y -110.8217,Z 141,A -122.4051,B 24.9628,C -1.4085,E1 24.9225,E2 568.7504} C_DIS
LIN {X -58.3856,Y -113.2528,Z 141,A -120.1206,B 24.963,C -1.4048,E1 24.9281,E2 566.4683} C_DIS
LIN {X -55.0813,Y -114.8944,Z 141,A -118.5842,B 24.9635,C -1.3968,E1 24.9319,E2 564.9468} C_DIS
LIN {X -47.3116,Y -118.3064,Z 141,A -114.6234,B 24.9633,C -1.3996,E1 24.9421,E2 560.9701} C_DIS
LIN {X -42.5885,Y -120.0889,Z 141,A -112.3816,B 24.9635,C -1.3961,E1 24.948,E2 558.7321} C_DIS
LIN {X -39.0905,Y -121.2713,Z 141,A -110.686,B 24.9635,C -1.3965,E1 24.9525,E2 557.0323} C_DIS
LIN {X -35.006,Y -122.5145,Z 141,A -108.8258,B 24.9637,C -1.3922,E1 24.9574,E2 555.1794} C_DIS
LIN {X -31.5384,Y -123.4507,Z 141,A -107.2683,B 24.9639,C -1.3884,E1 24.9616,E2 553.6285} C_DIS
LIN {X -28.052,Y -124.2896,Z 141,A -105.5062,B 24.9636,C -1.395,E1 24.9665,E2 551.8486} C_DIS
LIN {X -24.0563,Y -125.1241,Z 141,A -103.9112,B 24.9642,C -1.3823,E1 24.9708,E2 550.2819} C_DIS
LIN {X -21.0359,Y -125.6671,Z 141,A -102.4418,B 24.964,C -1.3862,E1 24.9748,E2 548.8016} C_DIS
LIN {X -17.8827,Y -126.1546,Z 141,A -100.9493,B 24.9639,C -1.3887,E1 24.979,E2 547.3019} C_DIS
LIN {X -13.3584,Y -126.7138,Z 141,A -98.5721,B 24.963,C -1.4048,E1 24.9857,E2 544.885} C_DIS
LIN {X -9.8724,Y -127.0339,Z 141,A -97.3399,B 24.9639,C -1.3876,E1 24.989,E2 543.6931} C_DIS
LIN {X -2.1614,Y -127.3975,Z 141,A -94.0563,B 24.9644,C -1.3785,E1 24.9981,E2 540.4305} C_DIS
LIN {X 0.8999,Y -127.3905,Z 141,A -92.6843,B 24.9644,C -1.3789,E1 25.002,E2 539.0576} C_DIS
Enddeposition()
LIN {X 0.8999,Y -127.3905,Z 141,A -92.6843,B 24.9644,C -1.3789,E1 25.002,E2 539.0576} C_DIS
Startdeposition()
$VEL.CP = VEL_PRINT
LIN {X 0.4082,Y -126.4436,Z 141,A -93.3053,B 24.8508,C -1.3516,E1 24.8853,E2 539.7273} C_DIS
LIN {X -2.8022,Y -126.4148,Z 141,A -95.4435,B 24.8525,C -1.3182,E1 24.8791,E2 541.9455} C_DIS
LIN {X -7.322,Y -126.2325,Z 141,A -96.7452,B 24.8507,C -1.3543,E1 24.8757,E2 543.1615} C_DIS
LIN {X -11.0231,Y -125.963,Z 141,A -98.5318,B 24.851,C -1.3492,E1 24.8707,E2 544.9609} C_DIS
LIN {X -14.6916,Y -125.5877,Z 141,A -100.3117,B 24.8512,C -1.3442,E1 24.8657,E2 546.754} C_DIS
LIN {X -18.6269,Y -125.0663,Z 141,A -102.1761,B 24.8514,C -1.3414,E1 24.8606,E2 548.6265} C_DIS
LIN {X -22.3565,Y -124.4516,Z 141,A -103.7392,B 24.851,C -1.3492,E1 24.8563,E2 550.1725} C_DIS
LIN {X -25.8968,Y -123.7653,Z 141,A -105.5341,B 24.8513,C -1.3421,E1 24.8513,E2 551.9864} C_DIS
LIN {X -30.7311,Y -122.6529,Z 141,A -107.4703,B 24.8505,C -1.3583,E1 24.8462,E2 553.8866} C_DIS
LIN {X -34.1977,Y -121.7313,Z 141,A -109.2594,B 24.8508,C -1.3515,E1 24.8413,E2 555.6947} C_DIS
LIN {X -37.4058,Y -120.7847,Z 141,A -110.7717,B 24.8508,C -1.3527,E1 24.8373,E2 557.2065} C_DIS
LIN {X -40.8577,Y -119.6619,Z 141,A -112.6217,B 24.8512,C -1.3443,E1 24.8323,E2 559.0802} C_DIS
LIN {X -45.1874,Y -118.0953,Z 141,A -114.8834,B 24.8515,C -1.338,E1 24.8263,E2 561.3616} C_DIS
LIN {X -48.2252,Y -116.8863,Z 141,A -116.4803,B 24.8517,C -1.3341,E1 24.8222,E2 562.9714} C_DIS
LIN {X -51.8045,Y -115.3441,Z 141,A -117.7919,B 24.8505,C -1.3575,E1 24.819,E2 564.2304} C_DIS
LIN {X -54.6356,Y -114.0303,Z 141,A -119.2198,B 24.8505,C -1.3585,E1 24.8153,E2 565.6594} C_DIS
LIN {X -58.0493,Y -112.3334,Z 141,A -121.5487,B 24.8518,C -1.3326,E1 24.8094,E2 568.0566} C_DIS
LIN {X -62.1233,Y -110.1324,Z 141,A -124.0791,B 24.8526,C -1.3156,E1 24.8031,E2 570.6351} C_DIS
LIN {X -67.9033,Y -106.6661,Z 141,A -126.0502,B 24.8499,C -1.3705,E1 24.7988,E2 572.4813} C_DIS
LIN {X -70.624,Y -104.8845,Z 141,A -127.7277,B 24.8502,C -1.3634,E1 24.7948,E2 574.1814} C_DIS
LIN {X -73.2609,Y -103.06,Z 141,A -129.1745,B 24.8501,C -1.3661,E1 24.7915,E2 575.6266} C_DIS
LIN {X -76.7261,Y -100.5063,Z 141,A -131.1079,B 24.8499,C -1.3704,E1 24.7872,E2 577.5567} C_DIS
LIN {X -80.1321,Y -97.8124,Z 141,A -133.0672,B 24.8497,C -1.3745,E1 24.7829,E2 579.5136} C_DIS
LIN {X -83.5204,Y -94.9359,Z 141,A -134.8592,B 24.8489,C -1.3888,E1 24.7792,E2 581.2786} C_DIS
LIN {X -85.884,Y -92.8036,Z 141,A -136.5649,B 24.8494,C -1.3795,E1 24.7756,E2 583.0133} C_DIS
LIN {X -88.9329,Y -89.8855,Z 141,A -138.4613,B 24.8491,C -1.3843,E1 24.7718,E2 584.9061} C_DIS
LIN {X -91.7776,Y -86.979,Z 141,A -140.3013,B 24.8489,C -1.3885,E1 24.7683,E2 586.744} C_DIS
LIN {X -94.7397,Y -83.7425,Z 141,A -141.9883,B 24.848,C -1.4069,E1 24.7652,E2 588.3946} C_DIS
LIN {X -96.6151,Y -81.5725,Z 141,A -143.6713,B 24.8487,C -1.3924,E1 24.762,E2 590.1201} C_DIS
LIN {X -99.2757,Y -78.3123,Z 141,A -145.5438,B 24.8484,C -1.3986,E1 24.7588,E2 591.9866} C_DIS
LIN {X -101.763,Y -75.0516,Z 141,A -147.3351,B 24.848,C -1.4063,E1 24.7558,E2 593.7682} C_DIS
LIN {X -104.4786,Y -71.2235,Z 141,A -149.588,B 24.848,C -1.406,E1 24.7522,E2 596.033} C_DIS
LIN {X -106.9606,Y -67.4376,Z 141,A -151.5799,B 24.8476,C -1.4141,E1 24.7492,E2 598.0156} C_DIS
LIN {X -109.2275,Y -63.7018,Z 141,A -153.6165,B 24.8474,C -1.4169,E1 24.7463,E2 600.0561} C_DIS
LIN {X -111.2868,Y -60.0308,Z 141,A -155.514,B 24.8471,C -1.4226,E1 24.7437,E2 601.9498} C_DIS
LIN {X -113.4447,Y -55.8411,Z 141,A -157.8205,B 24.8472,C -1.421,E1 24.7408,E2 604.2728} C_DIS
LIN {X -114.9476,Y -52.6799,Z 141,A -159.3347,B 24.8468,C -1.4288,E1 24.739,E2 605.7766} C_DIS
LIN {X -116.6476,Y -48.7985,Z 141,A -161.1057,B 24.8461,C -1.4411,E1 24.7371,E2 607.5279} C_DIS
LIN {X -117.8927,Y -45.7085,Z 141,A -162.6288,B 24.8459,C -1.445,E1 24.7355,E2 609.0503} C_DIS
LIN {X -119.0732,Y -42.5403,Z 141,A -164.1168,B 24.8456,C -1.4516,E1 24.7341,E2 610.531} C_DIS
LIN {X -120.0758,Y -39.6216,Z 141,A -165.6897,B 24.8458,C -1.448,E1 24.7327,E2 612.1215} C_DIS
LIN {X -122.2615,Y -32.2526,Z 141,A -169.056,B 24.8449,C -1.464,E1 24.7301,E2 615.4691} C_DIS
LIN {X -123.0009,Y -29.3065,Z 141,A -171.2116,B 24.8465,C -1.4336,E1 24.7287,E2 617.7102} C_DIS
LIN {X -124.1258,Y -24.1022,Z 141,A -172.7015,B 24.8439,C -1.4823,E1 24.7279,E2 619.0922} C_DIS
LIN {X -124.8989,Y -19.7081,Z 141,A -174.8687,B 24.8439,C -1.4823,E1 24.7269,E2 621.2726} C_DIS
LIN {X -125.3654,Y -16.4785,Z 141,A -176.4294,B 24.8438,C -1.4833,E1 24.7263,E2 622.84} C_DIS
LIN {X -125.8134,Y -12.6223,Z 141,A -178.2908,B 24.8438,C -1.4844,E1 24.7257,E2 624.71} C_DIS
LIN {X -126.1531,Y -8.5921,Z 141,A 179.8714,B 24.8434,C -1.4902,E1 24.7253,E2 626.5452} C_DIS
LIN {X -126.3547,Y -4.7522,Z 141,A 178.1973,B 24.8429,C -1.4989,E1 24.7251,E2 628.2084} C_DIS
LIN {X -126.4449,Y -0.5,Z 141,A 176.2535,B 24.8426,C -1.5045,E1 24.7251,E2 630.1507} C_DIS
LIN {X -126.3981,Y 3.4046,Z 141,A 174.4142,B 24.8425,C -1.5072,E1 24.7251,E2 631.9947} C_DIS
LIN {X -126.2113,Y 7.6667,Z 141,A 172.5251,B 24.842,C -1.5155,E1 24.7254,E2 633.8753} C_DIS
LIN {X -125.917,Y 11.5427,Z 141,A 170.6782,B 24.8419,C -1.5175,E1 24.7258,E2 635.7286} C_DIS
LIN {X -125.0608,Y 18.6627,Z 141,A 167.367,B 24.8414,C -1.5254,E1 24.727,E2 639.0408} C_DIS
LIN {X -124.4344,Y 22.4529,Z 141,A 165.7279,B 24.8408,C -1.5356,E1 24.7278,E2 640.6651} C_DIS
LIN {X -123.6501,Y 26.4332,Z 141,A 163.7554,B 24.8408,C -1.5356,E1 24.7289,E2 642.6493} C_DIS
LIN {X -122.6136,Y 30.8861,Z 141,A 161.7696,B 24.8402,C -1.5462,E1 24.7302,E2 644.6216} C_DIS
LIN {X -121.5813,Y 34.7343,Z 141,A 159.6318,B 24.8407,C -1.5372,E1 24.7318,E2 646.7935} C_DIS
LIN {X -120.6239,Y 37.9227,Z 141,A 158.3328,B 24.8399,C -1.5513,E1 24.7329,E2 648.0662} C_DIS
LIN {X -119.4185,Y 41.5597,Z 141,A 156.7197,B 24.8393,C -1.5623,E1 24.7343,E2 649.6621} C_DIS
LIN {X -118.0988,Y 45.1784,Z 141,A 154.6913,B 24.8397,C -1.5552,E1 24.7363,E2 651.7191} C_DIS
LIN {X -116.2723,Y 49.6888,Z 141,A 151.8034,B 24.841,C -1.5318,E1 24.7396,E2 654.6788} C_DIS
LIN {X -113.6716,Y 55.3813,Z 141,A 149.8541,B 24.8382,C -1.5797,E1 24.7418,E2 656.5243} C_DIS
LIN {X -110.9524,Y 60.6465,Z 141,A 146.9159,B 24.8384,C -1.5764,E1 24.7456,E2 659.4859} C_DIS
LIN {X -108.4274,Y 65.0542,Z 141,A 144.8667,B 24.8373,C -1.5945,E1 24.7485,E2 661.5027} C_DIS
LIN {X -106.3432,Y 68.4076,Z 141,A 142.9594,B 24.8373,C -1.5943,E1 24.7513,E2 663.4201} C_DIS
LIN {X -103.9695,Y 71.9641,Z 141,A 140.9919,B 24.8371,C -1.5985,E1 24.7544,E2 665.3875} C_DIS
LIN {X -101.4315,Y 75.4988,Z 141,A 139.1016,B 24.8366,C -1.6076,E1 24.7575,E2 667.2652} C_DIS
LIN {X -98.9989,Y 78.6615,Z 141,A 137.2159,B 24.8365,C -1.609,E1 24.7608,E2 669.1565} C_DIS
LIN {X -96.1412,Y 82.1302,Z 141,A 135.1536,B 24.8362,C -1.6132,E1 24.7645,E2 671.2183} C_DIS
LIN {X -93.257,Y 85.3909,Z 141,A 133.1732,B 24.8359,C -1.6179,E1 24.7682,E2 673.1963} C_DIS
LIN {X -89.6473,Y 89.1727,Z 141,A 131.0863,B 24.8348,C -1.6366,E1 24.7721,E2 675.2475} C_DIS
LIN {X -87.8135,Y 90.9793,Z 141,A 129.6539,B 24.8353,C -1.6274,E1 24.7751,E2 676.708} C_DIS
LIN {X -84.765,Y 93.8263,Z 141,A 127.3308,B 24.8363,C -1.6123,E1 24.7799,E2 679.0766} C_DIS
LIN {X -81.6793,Y 96.5242,Z 141,A 126.0756,B 24.8343,C -1.6438,E1 24.7825,E2 680.2615} C_DIS
LIN {X -79.6972,Y 98.1678,Z 141,A 124.6504,B 24.8349,C -1.6346,E1 24.7856,E2 681.714} C_DIS
LIN {X -76.1683,Y 100.9296,Z 141,A 122.6833,B 24.8345,C -1.6419,E1 24.7899,E2 683.6709} C_DIS
LIN {X -72.649,Y 103.4921,Z 141,A 120.6838,B 24.8343,C -1.6447,E1 24.7945,E2 685.6706} C_DIS
LIN {X -69.186,Y 105.8388,Z 141,A 118.7241,B 24.8343,C -1.6456,E1 24.799,E2 687.6348} C_DIS
LIN {X -65.3657,Y 108.2393,Z 141,A 116.1123,B 24.8356,C -1.6236,E1 24.8054,E2 690.3072} C_DIS
LIN {X -60.9281,Y 110.7985,Z 141,A 114.662,B 24.8329,C -1.6675,E1 24.8087,E2 691.6569} C_DIS
LIN {X -58.7353,Y 111.9736,Z 141,A 113.3393,B 24.8333,C -1.6605,E1 24.812,E2 693.0001} C_DIS
LIN {X -55.7383,Y 113.4955,Z 141,A 111.7939,B 24.8333,C -1.6619,E1 24.8159,E2 694.5462} C_DIS
LIN {X -51.1593,Y 115.6327,Z 141,A 109.5569,B 24.8328,C -1.6679,E1 24.8215,E2 696.7744} C_DIS
LIN {X -48.0828,Y 116.9465,Z 141,A 107.8866,B 24.8331,C -1.6629,E1 24.8259,E2 698.4605} C_DIS
LIN {X -43.7797,Y 118.6238,Z 141,A 105.8403,B 24.8328,C -1.6679,E1 24.8312,E2 700.4992} C_DIS
LIN {X -38.5044,Y 120.4383,Z 141,A 103.0275,B 24.8335,C -1.6578,E1 24.8387,E2 703.3413} C_DIS
LIN {X -35.2766,Y 121.4232,Z 141,A 101.8381,B 24.8324,C -1.6753,E1 24.8418,E2 704.491} C_DIS
LIN {X -31.4124,Y 122.48,Z 141,A 99.236,B 24.8345,C -1.6406,E1 24.8491,E2 707.1796} C_DIS
LIN {X -25.9751,Y 123.749,Z 141,A 97.5192,B 24.832,C -1.6807,E1 24.8535,E2 708.8031} C_DIS
LIN {X -22.981,Y 124.3399,Z 141,A 95.9742,B 24.8324,C -1.6742,E1 24.8578,E2 710.3653} C_DIS
LIN {X -19.2433,Y 124.9709,Z 141,A 94.3531,B 24.8321,C -1.68,E1 24.8622,E2 711.974} C_DIS
LIN {X -15.208,Y 125.5261,Z 141,A 92.4923,B 24.8321,C -1.6804,E1 24.8674,E2 713.8352} C_DIS
LIN {X -11.9275,Y 125.8801,Z 141,A 91.0047,B 24.832,C -1.6815,E1 24.8715,E2 715.321} C_DIS
LIN {X -7.8754,Y 126.1984,Z 141,A 89.165,B 24.832,C -1.6824,E1 24.8766,E2 717.1592} C_DIS
LIN {X -4.0606,Y 126.3799,Z 141,A 87.3984,B 24.832,C -1.6812,E1 24.8815,E2 718.929} C_DIS
LIN {X -0.4399,Y 126.4435,Z 141,A 85.6878,B 24.8322,C -1.6783,E1 24.8863,E2 720.6465} C_DIS
LIN {X 3.7057,Y 126.3898,Z 141,A 83.8419,B 24.8321,C -1.6801,E1 24.8915,E2 722.4878} C_DIS
LIN {X 7.7987,Y 126.2032,Z 141,A 82.0558,B 24.8318,C -1.6835,E1 24.8964,E2 724.2652} C_DIS
LIN {X 11.8854,Y 125.8841,Z 141,A 80.1836,B 24.8318,C -1.6827,E1 24.9017,E2 726.1384} C_DIS
LIN {X 15.2276,Y 125.5238,Z 141,A 78.6791,B 24.8318,C -1.6833,E1 24.9058,E2 727.6404} C_DIS
LIN {X 19.2343,Y 124.9723,Z 141,A 76.8483,B 24.8318,C -1.6829,E1 24.9109,E2 729.4705} C_DIS
LIN {X 22.8687,Y 124.36,Z 141,A 75.1041,B 24.8322,C -1.6786,E1 24.9157,E2 731.2229} C_DIS
LIN {X 27.8052,Y 123.3491,Z 141,A 73.1106,B 24.8313,C -1.6916,E1 24.9211,E2 733.183} C_DIS
LIN {X 32.3154,Y 122.2447,Z 141,A 70.7519,B 24.8322,C -1.6779,E1 24.9275,E2 735.5706} C_DIS
LIN {X 35.9945,Y 121.2131,Z 141,A 69.0807,B 24.8321,C -1.6796,E1 24.932,E2 737.2351} C_DIS
LIN {X 40.1147,Y 119.9116,Z 141,A 67.1031,B 24.8323,C -1.6771,E1 24.9373,E2 739.2149} C_DIS
LIN {X 44.962,Y 118.18,Z 141,A 64.4538,B 24.8334,C -1.6594,E1 24.9443,E2 741.9007} C_DIS
LIN {X 48.1797,Y 116.906,Z 141,A 63.1832,B 24.8326,C -1.6722,E1 24.9475,E2 743.1378} C_DIS
LIN {X 51.3874,Y 115.5307,Z 141,A 61.5834,B 24.8327,C -1.6696,E1 24.9516,E2 744.74} C_DIS
LIN {X 54.8712,Y 113.9177,Z 141,A 59.4725,B 24.834,C -1.6492,E1 24.957,E2 746.8938} C_DIS
LIN {X 58.3795,Y 112.1604,Z 141,A 58.3081,B 24.8323,C -1.677,E1 24.9597,E2 747.9889} C_DIS
LIN {X 60.9992,Y 110.7592,Z 141,A 56.2361,B 24.8346,C -1.6393,E1 24.965,E2 750.1443} C_DIS
LIN {X 64.9029,Y 108.5175,Z 141,A 54.7842,B 24.833,C -1.6653,E1 24.9684,E2 751.5302} C_DIS
LIN {X 67.9037,Y 106.6659,Z 141,A 53.0756,B 24.8335,C -1.6573,E1 24.9724,E2 753.2523} C_DIS
LIN {X 71.5279,Y 104.2697,Z 141,A 51.1379,B 24.8336,C -1.6555,E1 24.9769,E2 755.1877} C_DIS
LIN {X 74.6249,Y 102.0765,Z 141,A 49.416,B 24.8338,C -1.6524,E1 24.9808,E2 756.9109} C_DIS
LIN {X 79.1495,Y 98.6085,Z 141,A 46.7141,B 24.8345,C -1.6416,E1 24.9868,E2 759.6282} C_DIS
LIN {X 81.941,Y 96.3021,Z 141,A 45.2167,B 24.8342,C -1.6456,E1 24.99,E2 761.1104} C_DIS
LIN {X 85.251,Y 93.3853,Z 141,A 43.1858,B 24.8346,C -1.6399,E1 24.9942,E2 763.1467} C_DIS
LIN {X 88.393,Y 90.4164,Z 141,A 41.2606,B 24.8347,C -1.6374,E1 24.9981,E2 765.0698} C_DIS
LIN {X 91.424,Y 87.3502,Z 141,A 39.341,B 24.8349,C -1.6348,E1 25.0018,E2 766.9872} C_DIS
LIN {X 94.4389,Y 84.0823,Z 141,A 37.2967,B 24.8353,C -1.6287,E1 25.0056,E2 769.0369} C_DIS
LIN {X 97.2626,Y 80.7987,Z 141,A 35.3625,B 24.8355,C -1.6254,E1 25.0091,E2 770.9699} C_DIS
LIN {X 100.1663,Y 77.1703,Z 141,A 33.2384,B 24.8358,C -1.6193,E1 25.0128,E2 773.0985} C_DIS
LIN {X 103.2781,Y 72.952,Z 141,A 30.865,B 24.8362,C -1.6134,E1 25.0167,E2 775.4744} C_DIS
LIN {X 105.8831,Y 69.1179,Z 141,A 28.8211,B 24.8364,C -1.6108,E1 25.0198,E2 777.5143} C_DIS
LIN {X 108.1034,Y 65.5903,Z 141,A 26.3868,B 24.8383,C -1.578,E1 25.0235,E2 780.0137} C_DIS
LIN {X 110.5564,Y 61.3654,Z 141,A 24.7565,B 24.8369,C -1.6015,E1 25.0256,E2 781.5799} C_DIS
LIN {X 113.7697,Y 55.181,Z 141,A 21.5805,B 24.8375,C -1.5916,E1 25.0297,E2 784.7623} C_DIS
LIN {X 115.4639,Y 51.5367,Z 141,A 19.8706,B 24.8375,C -1.5921,E1 25.0316,E2 786.4619} C_DIS
LIN {X 116.966,Y 48.0361,Z 141,A 17.9674,B 24.8383,C -1.5778,E1 25.0337,E2 788.3882} C_DIS
LIN {X 118.744,Y 43.4533,Z 141,A 15.7208,B 24.8388,C -1.5702,E1 25.0359,E2 790.6404} C_DIS
LIN {X 121.0442,Y 36.5581,Z 141,A 12.3533,B 24.8396,C -1.5563,E1 25.0388,E2 794.0214} C_DIS
LIN {X 121.9874,Y 33.2804,Z 141,A 11.1951,B 24.8387,C -1.5714,E1 25.0396,E2 795.1373} C_DIS
LIN {X 122.9906,Y 29.3493,Z 141,A 9.3226,B 24.8392,C -1.5639,E1 25.0409,E2 797.0166} C_DIS
LIN {X 123.6692,Y 26.3448,Z 141,A 7.9953,B 24.8392,C -1.563,E1 25.0417,E2 798.3383} C_DIS
LIN {X 124.2956,Y 23.2142,Z 141,A 6.4697,B 24.8397,C -1.5543,E1 25.0425,E2 799.8755} C_DIS
LIN {X 124.9239,Y 19.5469,Z 141,A 4.8102,B 24.84,C -1.5503,E1 25.0433,E2 801.5348} C_DIS
LIN {X 125.4113,Y 16.1285,Z 141,A 3.1583,B 24.8405,C -1.5407,E1 25.0439,E2 803.1996} C_DIS
LIN {X 125.8866,Y 11.8603,Z 141,A 1.337,B 24.8405,C -1.5409,E1 25.0444,E2 805.0097} C_DIS
LIN {X 126.1957,Y 7.919,Z 141,A -0.4521,B 24.8409,C -1.5351,E1 25.0448,E2 806.8017} C_DIS
LIN {X 126.3749,Y 4.234,Z 141,A -2.217,B 24.8414,C -1.5248,E1 25.045,E2 808.5804} C_DIS
LIN {X 126.4478,Y 0.029,Z 141,A -4.2354,B 24.8421,C -1.5127,E1 25.045,E2 810.6155} C_DIS
LIN {X 126.3472,Y -4.9441,Z 141,A -6.4687,B 24.8425,C -1.5064,E1 25.0448,E2 812.8504} C_DIS
LIN {X 126.0925,Y -9.4219,Z 141,A -8.221,B 24.8421,C -1.5142,E1 25.0445,E2 814.5737} C_DIS
LIN {X 125.754,Y -13.1939,Z 141,A -9.9945,B 24.8425,C -1.5055,E1 25.044,E2 816.3571} C_DIS
LIN {X 125.3202,Y -16.8237,Z 141,A -11.725,B 24.8431,C -1.4962,E1 25.0434,E2 818.0993} C_DIS
LIN {X 124.6942,Y -20.9615,Z 141,A -13.4508,B 24.8429,C -1.4989,E1 25.0427,E2 819.8087} C_DIS
LIN {X 124.054,Y -24.4777,Z 141,A -15.7527,B 24.8452,C -1.4583,E1 25.0414,E2 822.1931} C_DIS
LIN {X 123.0169,Y -29.2401,Z 141,A -17.1078,B 24.8431,C -1.4952,E1 25.0406,E2 823.4529} C_DIS
LIN {X 122.1035,Y -32.8449,Z 141,A -19.0393,B 24.8442,C -1.477,E1 25.0392,E2 825.4164} C_DIS
LIN {X 120.3369,Y -38.8216,Z 141,A -21.7832,B 24.8444,C -1.472,E1 25.037,E2 828.1563} C_DIS
LIN {X 118.5169,Y -44.0658,Z 141,A -24.0461,B 24.8441,C -1.4772,E1 25.0349,E2 830.3942} C_DIS
LIN {X 116.9958,Y -47.9634,Z 141,A -26.363,B 24.8457,C -1.4493,E1 25.0325,E2 832.7642} C_DIS
LIN {X 115.1905,Y -52.1481,Z 141,A -28.5065,B 24.8462,C -1.4389,E1 25.03,E2 834.9206} C_DIS
LIN {X 113.8176,Y -55.0808,Z 141,A -29.6137,B 24.8455,C -1.453,E1 25.0288,E2 835.9884} C_DIS
LIN {X 112.4714,Y -57.7783,Z 141,A -30.9887,B 24.8457,C -1.4484,E1 25.027,E2 837.3669} C_DIS
LIN {X 110.8229,Y -60.8838,Z 141,A -32.6922,B 24.8463,C -1.4379,E1 25.0247,E2 839.0863} C_DIS
LIN {X 108.7233,Y -64.5576,Z 141,A -34.6105,B 24.8466,C -1.4322,E1 25.022,E2 841.0082} C_DIS
LIN {X 106.3621,Y -68.3781,Z 141,A -36.9756,B 24.8478,C -1.4094,E1 25.0184,E2 843.4154} C_DIS
LIN {X 104.2051,Y -71.6216,Z 141,A -38.4695,B 24.8474,C -1.4182,E1 25.0161,E2 844.8809} C_DIS
LIN {X 101.7281,Y -75.0991,Z 141,A -40.8197,B 24.8488,C -1.3916,E1 25.0122,E2 847.2829} C_DIS
LIN {X 98.8472,Y -78.8521,Z 141,A -42.3464,B 24.8474,C -1.4173,E1 25.0096,E2 848.7414} C_DIS
LIN {X 94.1685,Y -84.3843,Z 141,A -45.4443,B 24.8474,C -1.4181,E1 25.0041,E2 851.8233} C_DIS
LIN {X 92.1245,Y -86.6114,Z 141,A -47.5981,B 24.8497,C -1.3745,E1 24.9998,E2 854.0708} C_DIS
LIN {X 88.7371,Y -90.0789,Z 141,A -49.6911,B 24.8497,C -1.3744,E1 24.9956,E2 856.1554} C_DIS
LIN {X 85.5728,Y -93.0897,Z 141,A -51.1328,B 24.8485,C -1.3969,E1 24.9928,E2 857.5377} C_DIS
LIN {X 82.6479,Y -95.6962,Z 141,A -53.1151,B 24.8493,C -1.3822,E1 24.9886,E2 859.5469} C_DIS
LIN {X 79.6113,Y -98.2372,Z 141,A -54.8755,B 24.8493,C -1.3799,E1 24.9848,E2 861.3062} C_DIS
LIN {X 76.0728,Y -101.0017,Z 141,A -56.5348,B 24.8486,C -1.3946,E1 24.9812,E2 862.9246} C_DIS
LIN {X 73.0683,Y -103.1963,Z 141,A -58.8957,B 24.8506,C -1.3568,E1 24.9756,E2 865.3668} C_DIS
LIN {X 69.5409,Y -105.6052,Z 141,A -60.4135,B 24.8497,C -1.374,E1 24.9722,E2 866.8387} C_DIS
LIN {X 65.8331,Y -107.9561,Z 141,A -62.3995,B 24.8499,C -1.3703,E1 24.9675,E2 868.8272} C_DIS
LIN {X 62.0841,Y -110.1544,Z 141,A -64.277,B 24.8499,C -1.3713,E1 24.963,E2 870.6965} C_DIS
LIN {X 58.8585,Y -111.9089,Z 141,A -65.8796,B 24.8499,C -1.3715,E1 24.959,E2 872.294} C_DIS
LIN {X 55.9297,Y -113.4011,Z 141,A -67.3779,B 24.8499,C -1.3686,E1 24.9553,E2 873.7953} C_DIS
LIN {X 52.8695,Y -114.8599,Z 141,A -68.9503,B 24.8502,C -1.3643,E1 24.9513,E2 875.3738} C_DIS
LIN {X 48.3958,Y -116.8158,Z 141,A -71.1036,B 24.8502,C -1.3639,E1 24.9458,E2 877.5228} C_DIS
LIN {X 45.3322,Y -118.039,Z 141,A -72.7761,B 24.8508,C -1.3529,E1 24.9414,E2 879.2178} C_DIS
LIN {X 38.4743,Y -120.4479,Z 141,A -75.7059,B 24.8501,C -1.3668,E1 24.9338,E2 882.1086} C_DIS
LIN {X 33.5079,Y -121.9242,Z 141,A -78.2625,B 24.8507,C -1.3537,E1 24.9268,E2 884.692} C_DIS
LIN {X 29.8035,Y -122.8811,Z 141,A -80.02,B 24.8509,C -1.3507,E1 24.922,E2 886.4539} C_DIS
LIN {X 25.7502,Y -123.7951,Z 141,A -81.8994,B 24.8509,C -1.3491,E1 24.9169,E2 888.3346} C_DIS
LIN {X 22.3899,Y -124.4456,Z 141,A -83.3983,B 24.8509,C -1.3504,E1 24.9128,E2 889.8287} C_DIS
LIN {X 19.0436,Y -125.0018,Z 141,A -85.0538,B 24.8513,C -1.3434,E1 24.9082,E2 891.4993} C_DIS
LIN {X 15.0011,Y -125.5508,Z 141,A -86.7602,B 24.851,C -1.3493,E1 24.9035,E2 893.1905} C_DIS
LIN {X 11.6146,Y -125.9101,Z 141,A -88.3295,B 24.851,C -1.3471,E1 24.8991,E2 894.7638} C_DIS
LIN {X 7.5092,Y -126.221,Z 141,A -90.3882,B 24.8516,C -1.3368,E1 24.8933,E2 896.8461} C_DIS
LIN {X 3.5958,Y -126.3928,Z 141,A -92.2529,B 24.8518,C -1.3318,E1 24.8881,E2 898.7223} C_DIS
LIN {X 3.5958,Y -126.3928,Z 141,A -92.2529,B 24.8518,C -1.3318,E1 24.8881,E2 898.7223} C_DIS
Enddeposition()
LIN {X 0.8745,Y -125.4673,Z 141,A -92.5056,B 24.2837,C -1.2788,E1 24.3174,E2 899.025} C_DIS
Startdeposition()
$VEL.CP = VEL_PRINT
LIN {X 4.8992,Y -125.3764,Z 141,A -90.0935,B 24.2823,C -1.307,E1 24.3243,E2 896.5449} C_DIS
LIN {X 8.6508,Y -125.1743,Z 141,A -88.725,B 24.2831,C -1.2909,E1 24.328,E2 895.2161} C_DIS
LIN {X 12.5083,Y -124.848,Z 141,A -86.9307,B 24.2831,C -1.2932,E1 24.333,E2 893.4175} C_DIS
LIN {X 16.3838,Y -124.3976,Z 141,A -85.228,B 24.2831,C -1.2905,E1 24.3377,E2 891.7227} C_DIS
LIN {X 20.4281,Y -123.7979,Z 141,A -83.4353,B 24.2833,C -1.2882,E1 24.3426,E2 889.9373} C_DIS
LIN {X 23.5412,Y -123.2436,Z 141,A -81.9206,B 24.283,C -1.2928,E1 24.3468,E2 888.4131} C_DIS
LIN {X 27.5083,Y -122.42,Z 141,A -80.0446,B 24.2829,C -1.2958,E1 24.3519,E2 886.5325} C_DIS
LIN {X 30.8985,Y -121.6077,Z 141,A -78.5223,B 24.2829,C -1.294,E1 24.356,E2 885.0168} C_DIS
LIN {X 38.5511,Y -119.4031,Z 141,A -75.0551,B 24.2832,C -1.2898,E1 24.3653,E2 881.566} C_DIS
LIN {X 44.6057,Y -117.2768,Z 141,A -71.8778,B 24.2824,C -1.3056,E1 24.3737,E2 878.357} C_DIS
LIN {X 48.8117,Y -115.5888,Z 141,A -69.5864,B 24.2817,C -1.3196,E1 24.3797,E2 876.037} C_DIS
LIN {X 51.7444,Y -114.3064,Z 141,A -68.3093,B 24.282,C -1.3128,E1 24.3829,E2 874.78} C_DIS
LIN {X 55.2953,Y -112.6303,Z 141,A -66.6158,B 24.2821,C -1.3108,E1 24.3871,E2 873.0959} C_DIS
LIN {X 58.298,Y -111.1055,Z 141,A -65.1435,B 24.2821,C -1.3101,E1 24.3908,E2 871.6293} C_DIS
LIN {X 61.8588,Y -109.1659,Z 141,A -63.1483,B 24.2816,C -1.3205,E1 24.3957,E2 869.615} C_DIS
LIN {X 65.7268,Y -106.8811,Z 141,A -61.2125,B 24.2817,C -1.3186,E1 24.4003,E2 867.69} C_DIS
LIN {X 68.8246,Y -104.9132,Z 141,A -58.8151,B 24.2797,C -1.3581,E1 24.4061,E2 865.205} C_DIS
LIN {X 73.2348,Y -101.8839,Z 141,A -57.0675,B 24.2812,C -1.3282,E1 24.4099,E2 863.5362} C_DIS
LIN {X 76.4373,Y -99.5037,Z 141,A -55.3289,B 24.2812,C -1.3279,E1 24.4138,E2 861.8047} C_DIS
LIN {X 79.0373,Y -97.4515,Z 141,A -53.8089,B 24.2811,C -1.3317,E1 24.4171,E2 860.2816} C_DIS
LIN {X 84.2904,Y -92.9446,Z 141,A -50.8446,B 24.2811,C -1.3291,E1 24.4233,E2 857.3356} C_DIS
LIN {X 88.7804,Y -88.6664,Z 141,A -48.0551,B 24.281,C -1.3337,E1 24.4289,E2 854.5467} C_DIS
LIN {X 93.1228,Y -84.094,Z 141,A -45.0719,B 24.2803,C -1.3461,E1 24.4347,E2 851.547} C_DIS
LIN {X 96.9071,Y -79.7041,Z 141,A -42.3367,B 24.2797,C -1.3575,E1 24.4396,E2 848.797} C_DIS
LIN {X 100.5365,Y -75.0734,Z 141,A -39.6002,B 24.2792,C -1.3674,E1 24.4443,E2 846.0501} C_DIS
LIN {X 103.1956,Y -71.3748,Z 141,A -36.9992,B 24.2775,C -1.3997,E1 24.4486,E2 843.3839} C_DIS
LIN {X 105.7825,Y -67.481,Z 141,A -35.3902,B 24.2786,C -1.379,E1 24.4509,E2 841.8333} C_DIS
LIN {X 108.0389,Y -63.8064,Z 141,A -33.4283,B 24.2783,C -1.3844,E1 24.4537,E2 839.8688} C_DIS
LIN {X 110.1056,Y -60.1693,Z 141,A -31.5407,B 24.278,C -1.3889,E1 24.4563,E2 837.9804} C_DIS
LIN {X 111.7494,Y -57.0543,Z 141,A -30.0247,B 24.278,C -1.3891,E1 24.4582,E2 836.4723} C_DIS
LIN {X 115.0224,Y -50.1306,Z 141,A -26.6019,B 24.2777,C -1.3959,E1 24.4623,E2 833.0521} C_DIS
LIN {X 116.1709,Y -47.4103,Z 141,A -25.1767,B 24.2772,C -1.404,E1 24.4638,E2 831.6154} C_DIS
LIN {X 117.4337,Y -44.187,Z 141,A -23.6941,B 24.2772,C -1.404,E1 24.4653,E2 830.1414} C_DIS
LIN {X 119.2907,Y -38.9029,Z 141,A -20.9052,B 24.2761,C -1.4238,E1 24.4678,E2 827.3208} C_DIS
LIN {X 121.0505,Y -33.0218,Z 141,A -18.2076,B 24.2759,C -1.4273,E1 24.4699,E2 824.6304} C_DIS
LIN {X 122.5932,Y -26.7225,Z 141,A -15.3734,B 24.2758,C -1.4304,E1 24.4717,E2 821.8058} C_DIS
LIN {X 123.39,Y -22.7715,Z 141,A -13.4594,B 24.2752,C -1.4401,E1 24.4727,E2 819.8799} C_DIS
LIN {X 124.0512,Y -18.8317,Z 141,A -11.6387,B 24.2749,C -1.4459,E1 24.4735,E2 818.0562} C_DIS
LIN {X 124.5569,Y -15.1279,Z 141,A -10.0559,B 24.2749,C -1.4452,E1 24.4741,E2 816.4849} C_DIS
LIN {X 124.9237,Y -11.7202,Z 141,A -8.4191,B 24.2745,C -1.4539,E1 24.4745,E2 814.8369} C_DIS
LIN {X 125.2398,Y -7.6302,Z 141,A -6.7988,B 24.2748,C -1.4472,E1 24.4749,E2 813.2427} C_DIS
LIN {X 125.4177,Y -3.6988,Z 141,A -4.7425,B 24.2738,C -1.4663,E1 24.4751,E2 811.1529} C_DIS
LIN {X 125.4731,Y 0.4882,Z 141,A -2.8355,B 24.2734,C -1.4722,E1 24.4751,E2 809.2433} C_DIS
LIN {X 125.3813,Y 4.7736,Z 141,A -0.9805,B 24.2734,C -1.4734,E1 24.475,E2 807.3968} C_DIS
LIN {X 125.1631,Y 8.805,Z 141,A 0.8712,B 24.273,C -1.4798,E1 24.4746,E2 805.5409} C_DIS
LIN {X 124.8085,Y 12.8966,Z 141,A 2.7597,B 24.2726,C -1.4865,E1 24.4741,E2 803.6478} C_DIS
LIN {X 124.3833,Y 16.4934,Z 141,A 4.3793,B 24.2724,C -1.4901,E1 24.4736,E2 802.0293} C_DIS
LIN {X 123.7858,Y 20.501,Z 141,A 6.1558,B 24.2723,C -1.4923,E1 24.4728,E2 800.2583} C_DIS
LIN {X 123.2132,Y 23.7001,Z 141,A 7.6653,B 24.2719,C -1.4983,E1 24.472,E2 798.7435} C_DIS
LIN {X 122.3616,Y 27.7637,Z 141,A 9.5874,B 24.2715,C -1.5056,E1 24.4709,E2 796.8152} C_DIS
LIN {X 121.2022,Y 32.453,Z 141,A 12.3952,B 24.2693,C -1.5431,E1 24.4688,E2 793.9333} C_DIS
LIN {X 119.7691,Y 37.4035,Z 141,A 14.7331,B 24.2689,C -1.5495,E1 24.4669,E2 791.5937} C_DIS
LIN {X 118.185,Y 42.1383,Z 141,A 16.2097,B 24.2709,C -1.5156,E1 24.4656,E2 790.2078} C_DIS
LIN {X 117.0274,Y 45.2521,Z 141,A 18.0226,B 24.2698,C -1.535,E1 24.4638,E2 788.3582} C_DIS
LIN {X 115.3049,Y 49.4773,Z 141,A 19.914,B 24.27,C -1.5314,E1 24.4618,E2 786.4863} C_DIS
LIN {X 113.9486,Y 52.5248,Z 141,A 21.4066,B 24.2698,C -1.5343,E1 24.46,E2 784.9951} C_DIS
LIN {X 112.81,Y 54.931,Z 141,A 23.2582,B 24.2677,C -1.5699,E1 24.4577,E2 783.0675} C_DIS
LIN {X 110.5897,Y 59.2748,Z 141,A 24.8812,B 24.2691,C -1.5455,E1 24.4556,E2 781.5124} C_DIS
LIN {X 107.1284,Y 65.3237,Z 141,A 28.1085,B 24.2685,C -1.5564,E1 24.4511,E2 778.2759} C_DIS
LIN {X 104.9193,Y 68.8154,Z 141,A 29.9819,B 24.2682,C -1.5607,E1 24.4482,E2 776.4018} C_DIS
LIN {X 101.3828,Y 73.9272,Z 141,A 32.736,B 24.2681,C -1.5637,E1 24.4438,E2 773.6543} C_DIS
LIN {X 98.9752,Y 77.1205,Z 141,A 34.4698,B 24.2681,C -1.5637,E1 24.4409,E2 771.9292} C_DIS
LIN {X 96.6925,Y 79.9633,Z 141,A 36.2459,B 24.2675,C -1.5732,E1 24.4377,E2 770.1385} C_DIS
LIN {X 93.7618,Y 83.3812,Z 141,A 38.3344,B 24.2671,C -1.5796,E1 24.4339,E2 768.0441} C_DIS
LIN {X 90.811,Y 86.5849,Z 141,A 40.2658,B 24.267,C -1.5812,E1 24.4302,E2 766.1175} C_DIS
LIN {X 87.8411,Y 89.5964,Z 141,A 42.1634,B 24.2668,C -1.5837,E1 24.4265,E2 764.2222} C_DIS
LIN {X 84.708,Y 92.5646,Z 141,A 44.1566,B 24.2665,C -1.5889,E1 24.4224,E2 762.2248} C_DIS
LIN {X 81.5512,Y 95.3578,Z 141,A 45.9635,B 24.2666,C -1.5869,E1 24.4186,E2 760.43} C_DIS
LIN {X 77.0803,Y 99.0064,Z 141,A 48.7075,B 24.266,C -1.5972,E1 24.4126,E2 757.6716} C_DIS
LIN {X 73.6204,Y 101.6052,Z 141,A 50.4488,B 24.2665,C -1.5893,E1 24.4087,E2 755.956} C_DIS
LIN {X 70.7976,Y 103.5922,Z 141,A 52.1745,B 24.2659,C -1.5993,E1 24.4047,E2 754.2122} C_DIS
LIN {X 67.3407,Y 105.8723,Z 141,A 54.1559,B 24.2654,C -1.6067,E1 24.4001,E2 752.2194} C_DIS
LIN {X 63.6444,Y 108.1341,Z 141,A 56.7341,B 24.2634,C -1.6391,E1 24.3937,E2 749.5709} C_DIS
LIN {X 59.0486,Y 110.7113,Z 141,A 58.3885,B 24.2655,C -1.6056,E1 24.3899,E2 748.0026} C_DIS
LIN {X 54.2255,Y 113.1491,Z 141,A 60.8273,B 24.2654,C -1.6074,E1 24.3838,E2 745.5662} C_DIS
LIN {X 51.3813,Y 114.4688,Z 141,A 62.2906,B 24.2652,C -1.6106,E1 24.38,E2 744.099} C_DIS
LIN {X 48.3247,Y 115.7922,Z 141,A 63.7728,B 24.2652,C -1.6104,E1 24.3762,E2 742.6208} C_DIS
LIN {X 43.1505,Y 117.82,Z 141,A 66.4301,B 24.2647,C -1.6186,E1 24.3693,E2 739.9495} C_DIS
LIN {X 39.9286,Y 118.9493,Z 141,A 67.9369,B 24.2647,C -1.6175,E1 24.3653,E2 738.4485} C_DIS
LIN {X 37.0284,Y 119.8839,Z 141,A 69.1668,B 24.2652,C -1.6109,E1 24.3621,E2 737.237} C_DIS
LIN {X 33.1284,Y 121.0212,Z 141,A 71.2267,B 24.2645,C -1.622,E1 24.3565,E2 735.1538} C_DIS
LIN {X 29.5291,Y 121.9476,Z 141,A 72.6275,B 24.2653,C -1.6089,E1 24.3528,E2 733.7869} C_DIS
LIN {X 26.1744,Y 122.7117,Z 141,A 74.5365,B 24.2642,C -1.6258,E1 24.3475,E2 731.8396} C_DIS
LIN {X 22.1957,Y 123.4931,Z 141,A 76.2631,B 24.2645,C -1.6206,E1 24.3428,E2 730.1275} C_DIS
LIN {X 18.4803,Y 124.1056,Z 141,A 78.0496,B 24.2643,C -1.6243,E1 24.3378,E2 728.3338} C_DIS
LIN {X 14.8764,Y 124.5869,Z 141,A 79.6418,B 24.2645,C -1.6215,E1 24.3334,E2 726.7498} C_DIS
LIN {X 11.2387,Y 124.9695,Z 141,A 81.436,B 24.2641,C -1.6275,E1 24.3284,E2 724.9421} C_DIS
LIN {X 7.2917,Y 125.2607,Z 141,A 83.2035,B 24.2642,C -1.6257,E1 24.3235,E2 723.1797} C_DIS
LIN {X 3.3783,Y 125.4266,Z 141,A 84.9313,B 24.2644,C -1.6227,E1 24.3187,E2 721.4596} C_DIS
LIN {X -0.5456,Y 125.471,Z 141,A 86.6837,B 24.2645,C -1.6205,E1 24.3138,E2 719.7127} C_DIS
LIN {X -4.1697,Y 125.4046,Z 141,A 88.4787,B 24.2642,C -1.6266,E1 24.3088,E2 717.9027} C_DIS
LIN {X -8.0691,Y 125.2128,Z 141,A 90.2272,B 24.2643,C -1.6243,E1 24.3039,E2 716.1591} C_DIS
LIN {X -12.038,Y 124.8932,Z 141,A 91.9438,B 24.2647,C -1.6188,E1 24.2992,E2 714.4552} C_DIS
LIN {X -15.588,Y 124.5018,Z 141,A 93.7103,B 24.2643,C -1.6241,E1 24.2942,E2 712.6745} C_DIS
LIN {X -19.5318,Y 123.9428,Z 141,A 95.5347,B 24.2643,C -1.6231,E1 24.2892,E2 710.8508} C_DIS
LIN {X -23.5214,Y 123.2474,Z 141,A 97.279,B 24.2648,C -1.6169,E1 24.2844,E2 709.1199} C_DIS
LIN {X -26.3368,Y 122.6766,Z 141,A 99.9182,B 24.2609,C -1.6775,E1 24.2769,E2 706.3296} C_DIS
LIN {X -34.353,Y 120.6787,Z 141,A 102.2116,B 24.2655,C -1.6049,E1 24.2712,E2 704.2095} C_DIS
LIN {X -41.5877,Y 118.3801,Z 141,A 105.7951,B 24.2655,C -1.606,E1 24.2616,E2 700.6166} C_DIS
LIN {X -45.5884,Y 116.8967,Z 141,A 107.7574,B 24.2655,C -1.6041,E1 24.2565,E2 698.6549} C_DIS
LIN {X -48.6706,Y 115.6477,Z 141,A 109.3875,B 24.2654,C -1.607,E1 24.2522,E2 697.0139} C_DIS
LIN {X -52.1435,Y 114.1249,Z 141,A 111.0912,B 24.2656,C -1.6031,E1 24.2479,E2 695.3155} C_DIS
LIN {X -56.2647,Y 112.1513,Z 141,A 113.2551,B 24.2656,C -1.6031,E1 24.2425,E2 693.1454} C_DIS
LIN {X -59.0973,Y 110.6851,Z 141,A 115.1328,B 24.2646,C -1.6198,E1 24.2377,E2 691.2216} C_DIS
LIN {X -62.7689,Y 108.6441,Z 141,A 116.6077,B 24.2661,C -1.5963,E1 24.2343,E2 689.7996} C_DIS
LIN {X -66.5624,Y 106.3631,Z 141,A 118.672,B 24.2661,C -1.5945,E1 24.2294,E2 687.7333} C_DIS
LIN {X -70.123,Y 104.05,Z 141,A 120.6236,B 24.2664,C -1.5912,E1 24.2248,E2 685.7828} C_DIS
LIN {X -73.8509,Y 101.4381,Z 141,A 122.6426,B 24.2668,C -1.5843,E1 24.2202,E2 683.7736} C_DIS
LIN {X -77.1705,Y 98.9365,Z 141,A 124.6367,B 24.2668,C -1.5845,E1 24.2158,E2 681.7714} C_DIS
LIN {X -80.2442,Y 96.46,Z 141,A 126.8569,B 24.2659,C -1.5993,E1 24.2109,E2 679.5066} C_DIS
LIN {X -83.5157,Y 93.6417,Z 141,A 128.415,B 24.2673,C -1.5762,E1 24.2078,E2 677.9985} C_DIS
LIN {X -86.8727,Y 90.536,Z 141,A 130.4931,B 24.2676,C -1.5708,E1 24.2036,E2 675.9247} C_DIS
LIN {X -89.0652,Y 88.3796,Z 141,A 132.0666,B 24.2674,C -1.5749,E1 24.2004,E2 674.3343} C_DIS
LIN {X -92.6629,Y 84.6008,Z 141,A 134.3023,B 24.2681,C -1.5623,E1 24.1962,E2 672.1193} C_DIS
LIN {X -95.4827,Y 81.4042,Z 141,A 136.2614,B 24.2684,C -1.5578,E1 24.1926,E2 670.1619} C_DIS
LIN {X -98.3702,Y 77.8908,Z 141,A 138.3602,B 24.2687,C -1.5533,E1 24.189,E2 668.0641} C_DIS
LIN {X -100.9657,Y 74.4954,Z 141,A 140.299,B 24.269,C -1.5474,E1 24.1857,E2 666.13} C_DIS
LIN {X -103.3129,Y 71.2045,Z 141,A 142.1846,B 24.2692,C -1.544,E1 24.1827,E2 664.2432} C_DIS
LIN {X -105.8723,Y 67.3407,Z 141,A 144.3235,B 24.2695,C -1.539,E1 24.1795,E2 662.1054} C_DIS
LIN {X -107.6033,Y 64.5385,Z 141,A 145.7814,B 24.2699,C -1.5326,E1 24.1774,E2 660.6553} C_DIS
LIN {X -110.127,Y 60.13,Z 141,A 148.291,B 24.2699,C -1.5342,E1 24.1739,E2 658.1285} C_DIS
LIN {X -112.3432,Y 55.8772,Z 141,A 150.244,B 24.2708,C -1.5172,E1 24.1715,E2 656.2061} C_DIS
LIN {X -115.3386,Y 49.3995,Z 141,A 153.4535,B 24.2715,C -1.5051,E1 24.1678,E2 653.0082} C_DIS
LIN {X -116.6977,Y 46.098,Z 141,A 155.2531,B 24.2714,C -1.5074,E1 24.1659,E2 651.1924} C_DIS
LIN {X -118.0332,Y 42.5592,Z 141,A 156.911,B 24.2719,C -1.499,E1 24.1643,E2 649.5454} C_DIS
LIN {X -118.9136,Y 40.0357,Z 141,A 158.5047,B 24.2712,C -1.5115,E1 24.1628,E2 647.9118} C_DIS
LIN {X -119.9516,Y 36.807,Z 141,A 159.6677,B 24.2724,C -1.4897,E1 24.1619,E2 646.7953} C_DIS
LIN {X -120.8279,Y 33.8198,Z 141,A 161.121,B 24.2726,C -1.4865,E1 24.1608,E2 645.3409} C_DIS
LIN {X -121.6985,Y 30.5407,Z 141,A 162.821,B 24.2726,C -1.4882,E1 24.1596,E2 643.6268} C_DIS
LIN {X -122.7101,Y 26.1817,Z 141,A 164.8795,B 24.2729,C -1.4822,E1 24.1584,E2 641.5703} C_DIS
LIN {X -123.496,Y 22.1795,Z 141,A 166.625,B 24.2735,C -1.4711,E1 24.1575,E2 639.8415} C_DIS
LIN {X -124.5347,Y 15.3135,Z 141,A 169.826,B 24.274,C -1.462,E1 24.1562,E2 636.6429} C_DIS
LIN {X -124.9169,Y 11.7904,Z 141,A 171.5211,B 24.2741,C -1.4601,E1 24.1557,E2 634.942} C_DIS
LIN {X -125.2296,Y 7.7953,Z 141,A 173.3197,B 24.2745,C -1.4528,E1 24.1554,E2 633.1502} C_DIS
LIN {X -125.4188,Y 3.6594,Z 141,A 175.2317,B 24.2748,C -1.4475,E1 24.1552,E2 631.2392} C_DIS
LIN {X -125.4747,Y -0.219,Z 141,A 177.1081,B 24.2748,C -1.4463,E1 24.1552,E2 629.3541} C_DIS
LIN {X -125.4057,Y -4.131,Z 141,A 178.9002,B 24.2752,C -1.4407,E1 24.1552,E2 627.5644} C_DIS
LIN {X -125.2266,Y -7.8453,Z 141,A -179.494,B 24.2757,C -1.4312,E1 24.1555,E2 625.9719} C_DIS
LIN {X -124.9072,Y -11.8916,Z 141,A -177.611,B 24.276,C -1.4265,E1 24.156,E2 624.0888} C_DIS
LIN {X -124.4617,Y -15.8949,Z 141,A -175.7469,B 24.2763,C -1.4217,E1 24.1566,E2 622.225} C_DIS
LIN {X -124.0529,Y -18.8203,Z 141,A -174.3007,B 24.2763,C -1.4217,E1 24.1572,E2 620.7699} C_DIS
LIN {X -123.2082,Y -23.7265,Z 141,A -172.08,B 24.2768,C -1.4121,E1 24.1583,E2 618.559} C_DIS
LIN {X -122.0211,Y -29.224,Z 141,A -169.5567,B 24.2773,C -1.4021,E1 24.1598,E2 616.045} C_DIS
LIN {X -121.2048,Y -32.4433,Z 141,A -167.3986,B 24.276,C -1.4258,E1 24.1614,E2 613.8159} C_DIS
LIN {X -119.8913,Y -37.004,Z 141,A -165.7563,B 24.2777,C -1.3958,E1 24.1627,E2 612.2371} C_DIS
LIN {X -118.5889,Y -40.9856,Z 141,A -163.896,B 24.2781,C -1.3877,E1 24.1644,E2 610.3857} C_DIS
LIN {X -117.2298,Y -44.7313,Z 141,A -161.9392,B 24.2781,C -1.3883,E1 24.1663,E2 608.4159} C_DIS
LIN {X -115.8308,Y -48.2323,Z 141,A -160.35,B 24.2787,C -1.3775,E1 24.1679,E2 606.8442} C_DIS
LIN {X -114.5746,Y -51.1446,Z 141,A -158.8797,B 24.2788,C -1.3742,E1 24.1696,E2 605.3735} C_DIS
LIN {X -113.3221,Y -53.8635,Z 141,A -157.0992,B 24.2781,C -1.3887,E1 24.1718,E2 603.5475} C_DIS
LIN {X -111.6634,Y -57.2232,Z 141,A -155.7081,B 24.2791,C -1.3696,E1 24.1735,E2 602.1954} C_DIS
LIN {X -109.5422,Y -61.1898,Z 141,A -153.6083,B 24.2793,C -1.366,E1 24.1763,E2 600.0932} C_DIS
LIN {X -107.2618,Y -65.104,Z 141,A -151.5595,B 24.2796,C -1.3595,E1 24.1792,E2 598.0493} C_DIS
LIN {X -105.2212,Y -68.3526,Z 141,A -149.9161,B 24.2801,C -1.3501,E1 24.1817,E2 596.4203} C_DIS
LIN {X -103.65,Y -70.7131,Z 141,A -148.3544,B 24.2797,C -1.3587,E1 24.1842,E2 594.8296} C_DIS
LIN {X -100.8609,Y -74.6377,Z 141,A -146.2478,B 24.2802,C -1.349,E1 24.1876,E2 592.736} C_DIS
LIN {X -98.207,Y -78.0958,Z 141,A -144.2834,B 24.2805,C -1.343,E1 24.191,E2 590.7768} C_DIS
LIN {X -95.373,Y -81.5333,Z 141,A -142.5105,B 24.2813,C -1.3264,E1 24.1941,E2 589.0359} C_DIS
LIN {X -93.2078,Y -84.0002,Z 141,A -140.7133,B 24.2808,C -1.3364,E1 24.1975,E2 587.206} C_DIS
LIN {X -90.2715,Y -87.1473,Z 141,A -138.7446,B 24.281,C -1.3322,E1 24.2013,E2 585.2388} C_DIS
LIN {X -87.1292,Y -90.2891,Z 141,A -136.7281,B 24.2813,C -1.3273,E1 24.2053,E2 583.2254} C_DIS
LIN {X -84.0829,Y -93.1329,Z 141,A -134.7581,B 24.2813,C -1.3265,E1 24.2094,E2 581.2493} C_DIS
LIN {X -80.6833,Y -96.0926,Z 141,A -132.7458,B 24.2816,C -1.3204,E1 24.2136,E2 579.2439} C_DIS
LIN {X -77.3565,Y -98.7905,Z 141,A -130.7785,B 24.2818,C -1.3172,E1 24.2179,E2 577.2766} C_DIS
LIN {X -73.9276,Y -101.3825,Z 141,A -128.8356,B 24.282,C -1.3129,E1 24.2223,E2 575.3373} C_DIS
LIN {X -71.1165,Y -103.3733,Z 141,A -127.2203,B 24.282,C -1.3122,E1 24.226,E2 573.7181} C_DIS
LIN {X -67.3159,Y -105.8881,Z 141,A -125.3435,B 24.2827,C -1.2995,E1 24.2303,E2 571.8659} C_DIS
LIN {X -62.4232,Y -108.844,Z 141,A -122.5486,B 24.2825,C -1.3041,E1 24.2371,E2 569.051} C_DIS
LIN {X -60.0245,Y -110.1846,Z 141,A -121.0631,B 24.282,C -1.313,E1 24.2408,E2 567.5393} C_DIS
LIN {X -55.7487,Y -112.4066,Z 141,A -119.098,B 24.2827,C -1.2993,E1 24.2456,E2 565.6022} C_DIS
LIN {X -52.6325,Y -113.8988,Z 141,A -117.5808,B 24.2829,C -1.2946,E1 24.2494,E2 564.0925} C_DIS
LIN {X -50.0965,Y -115.0372,Z 141,A -115.7646,B 24.2817,C -1.3187,E1 24.2542,E2 562.213} C_DIS
LIN {X -46.0964,Y -116.6991,Z 141,A -114.211,B 24.2828,C -1.2969,E1 24.2581,E2 560.7093} C_DIS
LIN {X -42.8089,Y -117.9432,Z 141,A -112.6362,B 24.283,C -1.294,E1 24.2622,E2 559.1382} C_DIS
LIN {X -39.3125,Y -119.1544,Z 141,A -110.9038,B 24.283,C -1.2946,E1 24.2668,E2 557.401} C_DIS
LIN {X -35.3204,Y -120.3977,Z 141,A -109.1053,B 24.2833,C -1.288,E1 24.2716,E2 555.6154} C_DIS
LIN {X -31.4344,Y -121.4717,Z 141,A -107.0931,B 24.2829,C -1.2949,E1 24.2771,E2 553.5833} C_DIS
LIN {X -26.8884,Y -122.5576,Z 141,A -105.0555,B 24.2832,C -1.2892,E1 24.2826,E2 551.5567} C_DIS
LIN {X -23.3598,Y -123.2783,Z 141,A -103.4344,B 24.2832,C -1.2875,E1 24.287,E2 549.938} C_DIS
LIN {X -19.3779,Y -123.9666,Z 141,A -101.5825,B 24.2833,C -1.2872,E1 24.2921,E2 548.0849} C_DIS
LIN {X -15.3463,Y -124.5308,Z 141,A -99.6805,B 24.2833,C -1.2889,E1 24.2974,E2 546.1775} C_DIS
LIN {X -11.3984,Y -124.9546,Z 141,A -97.753,B 24.283,C -1.2941,E1 24.3028,E2 544.236} C_DIS
LIN {X -7.2753,Y -125.2617,Z 141,A -96.1852,B 24.2837,C -1.2789,E1 24.3071,E2 542.7047} C_DIS
LIN {X -3.289,Y -125.4291,Z 141,A -94.2654,B 24.2835,C -1.2838,E1 24.3125,E2 540.7728} C_DIS
LIN {X 0.8745,Y -125.4673,Z 141,A -92.5025,B 24.2838,C -1.2776,E1 24.3174,E2 539.025} C_DIS
Enddeposition()
LIN {X 0.8745,Y -125.4673,Z 141,A -92.5025,B 24.2838,C -1.2776,E1 24.3174,E2 539.025} C_DIS
Startdeposition()
$VEL.CP = VEL_PRINT
LIN {X -0.5312,Y -124.4992,Z 141,A -93.4462,B 23.6888,C -1.1611,E1 23.7144,E2 540.1744} C_DIS
LIN {X -3.7759,Y -124.4433,Z 141,A -94.975,B 23.6889,C -1.1593,E1 23.7102,E2 541.708} C_DIS
LIN {X -6.6709,Y -124.322,Z 141,A -96.2616,B 23.6889,C -1.1613,E1 23.7066,E2 542.9898} C_DIS
LIN {X -9.9693,Y -124.1014,Z 141,A -97.7517,B 23.6888,C -1.1628,E1 23.7024,E2 544.4769} C_DIS
LIN {X -13.2434,Y -123.7937,Z 141,A -99.3907,B 23.689,C -1.1572,E1 23.6978,E2 546.1307} C_DIS
Enddeposition()
END
